// TIA Portal V17 program export: 1 tag tables, 0 data types, 2 data blocks, 7 code blocks (in call order from the OBs), 24 instance data blocks

VAR_GLOBAL   // PLC tag table "Default tag table"
   i_PB_RESET_BEZPIECZENSTWA AT %I0.0 : Bool;
   i_KURTYNA_ŚWIETLNA_OK AT %I0.1 : Bool;
   i_E_STOP_OK AT %I0.2 : Bool;
   i_PB_START AT %I0.3 : Bool;
   i_PB_STOP AT %I0.4 : Bool;
   i_SIŁOWNIK_ZACISKAJĄCY_UGÓRY AT %I0.5 : Bool;
   i_SIŁOWNIK_ZACISKAJĄCY_W_DOLE AT %I0.6 : Bool;
   "i_SIŁOWNIK NASTAWY_GŁĘBOKIE" AT %I0.7 : Bool;
   "i_SIŁOWNIK NASTAWY _PŁYTKIE" AT %I1.0 : Bool;
   i_SIŁOWNIK_ODBIORU_POZ_STÓŁ AT %I1.1 : Bool;
   i_SIŁOWNIK_ODBIORU_POZ_ZRZUT AT %I1.2 : Bool;
   i_CZUJNIK_POZYCJI_STOŁU AT %I1.3 : Bool;
   i_CZUJNIK_SZTUKI_OK AT %I1.4 : Bool;
   i_CZUJNIK_PŁYTKIE_PRZÓD AT %I1.5 : Bool;
   Axis_1_Drive_IN AT %I68.0 : "PD_TEL3_IN";
   q_GŁÓWNY_ZAWÓR_POWIETRZA_ON AT %Q0.0 : Bool;
   q_NIEBIESKA_LAMPKA_SAFETY AT %Q0.1 : Bool;
   q_SIŁOWNIK_ZACISKAJĄCY_DOL AT %Q0.2 : Bool;
   q_EJECTOR_VACUM AT %Q0.3 : Bool;
   q_SIŁOWNIK_ZMIANY_GŁĘBOKIE AT %Q0.4 : Bool;
   q_EJECTOR_BLOWOFF AT %Q0.5 : Bool;
   q_SIŁOWNIK_ODBIERAJĄCY_STÓŁ AT %Q0.6 : Bool;
   q_LED_LAMP AT %Q0.7 : Bool;
   q_REZERWA1 AT %Q1.0 : Bool;
   q_REZERWA2 AT %Q1.1 : Bool;
   q_CZERWONA_KOLUMNA_SYGNALIZACYJNA AT %Q8.0 : Bool;
   q_ZÓŁTA_KOLUMNA_SYGNALIZACYJNA AT %Q8.1 : Bool;
   q_ZIELONA_KOLUMNA_SYGNALIZACYJNA AT %Q8.2 : Bool;
   q_BUZZER_KOLUMNA_SYGNALIZACYJNA AT %Q8.3 : Bool;
   q_SAFETY_RELAY_RESET AT %Q8.4 : Bool;
   q_REZERWA4 AT %Q8.5 : Bool;
   q_REZERWA5 AT %Q8.6 : Bool;
   q_REZERWA6 AT %Q8.7 : Bool;
   Clock_Byte AT %MB0 : Byte;
   Clock_10Hz AT %M0.0 : Bool;
   Clock_5Hz AT %M0.1 : Bool;
   "Clock_2.5Hz" AT %M0.2 : Bool;
   Clock_2Hz AT %M0.3 : Bool;
   "Clock_1.25Hz" AT %M0.4 : Bool;
   Clock_1Hz AT %M0.5 : Bool;
   "Clock_0.625Hz" AT %M0.6 : Bool;
   "Clock_0.5Hz" AT %M0.7 : Bool;
   m_SAFETY_OK AT %M1.0 : Bool;
   m_AUTO_MODE AT %M1.1 : Bool;
   m_SERVO_READY AT %M1.2 : Bool;
   MAN_SIŁ_ZAG_GÓRA AT %M1.3 : Bool;
   MAN_SIŁ_ZAG_DÓŁ AT %M1.4 : Bool;
   MAN_SIŁ_NASTAWY_GŁĘBOKIE AT %M1.5 : Bool;
   MAN_SIŁ_NASTAWY_PŁYTKIE AT %M1.6 : Bool;
   MAN_SIŁ_ODBIOR_STÓŁ AT %M1.7 : Bool;
   MAN_SIŁ_ODBIOR_ZRZUT AT %M2.0 : Bool;
   MAN_JOG_STOL_FWD AT %M2.1 : Bool;
   MAN_JOG_STOL_BWD AT %M2.2 : Bool;
   MAN_POZYCJA_STÓŁ_FWD AT %M2.3 : Bool;
   MAN_POZYCJA_STÓŁ_BWD AT %M2.4 : Bool;
   MAN_EJECTOR_SSANIE AT %M2.5 : Bool;
   MAN_EJECTOR_PRZEDMUCH AT %M2.6 : Bool;
   TP_ZAPISZ_WARTOŚĆ_PRED AT %M2.7 : Bool;
   TP_ZAPISZ_WARTOŚĆ_CZASU_PRZEDMUCHU AT %M3.0 : Bool;
   TP_ZAPISZ_WARTOSC_CZASU_SSANIA AT %M3.1 : Bool;
   TP_AKT_PRED_STOŁU AT %MW4 : Int;
   TP_NOWA_PRED_STOŁU AT %MW6 : Int;
   TP_AKT_CZAS_PRZEDMUCHU AT %MD50 : DInt;
   TP_NOWY_CZAS_PRZEDMUCHU AT %MD54 : DInt;
   TP_AKT_CZAS_SSANIA AT %MD58 : DInt;
   TP_NOWY_CZAS_SSANIA AT %MD62 : DInt;
   TP_LICZNIK_CAŁKOWITY AT %MD16 : DInt;
   TP_LICZNIK_ZADANE AT %MD20 : DInt;
   TP_LICZNIK_WYKONANE AT %MD24 : DInt;
   TP_KASUJ_LICZNIK_ZADANE AT %M3.2 : Bool;
   TP_USTAW_LICZNIK_ZADANE AT %M3.3 : Bool;
   TP_KASUJ_LICZNIK_AKTUALNE AT %M3.4 : Bool;
   m_STOL_KAT_OBROTU AT %MW28 : Int;
   TP_LED_ZAŁĄCZ AT %M3.5 : Bool;
   m_SRV_STO_ON AT %M3.6 : Bool;
   TP_USTAW_CZAS_TAKTU AT %M3.7 : Bool;
   AUTO_NUMER_KROKU AT %MW30 : Int;
   AUTO_KROK_1_ZAŁADUNEK AT %M32.0 : Bool;
   AUTO_KROK_2_OBRÓT_USTAW_GŁĘBOKIE AT %M32.1 : Bool;
   AUTO_KROK_3_ROZŁADUNEK AT %M32.2 : Bool;
   AUTO_KROK_4_ZJAZD_GŁĘBOKIE AT %M32.3 : Bool;
   AUTO_KROK_5_OBRÓT_USTAW_PLYTKIE AT %M32.4 : Bool;
   "AUTO_KROK_6_ZJAZD GŁOWICY PŁYTKIE" AT %M32.5 : Bool;
   AUTO_SERVO_FWD AT %M34.0 : Bool;
   AUTO_SIŁOWNIK_ZACISKAJĄCY_DÓŁ AT %M34.1 : Bool;
   AUTO_SIŁOWNIK_ZACISKAJĄCY_GÓRA AT %M34.2 : Bool;
   AUTO_SIŁOWNIK_NASTAWY_GŁĘBOKIE AT %M34.3 : Bool;
   AUTO_SIŁOWNIK_NASTAWY_PŁYTKIE AT %M34.4 : Bool;
   AUTO_SIŁOWNIK_ODBIORU_STÓŁ AT %M34.5 : Bool;
   AUTO_SIŁOWNIK_ODBIORU_ZRZUT AT %M34.6 : Bool;
   AUTO_EJECTOR_SSANIE AT %M34.7 : Bool;
   AUTO_EJECTOR_PRZEDMUCH AT %M35.0 : Bool;
   AUTO_TAKT_OBRÓT AT %MW38 : Int;
   TP_TAKT_ZADANA AT %MW40 : Int;
   TEST_BIT AT %M100.2 : Bool;
   TP_LAMP_TEST AT %M43.1 : Bool;
   m_TRYB_RĘCZNY_MOŻLIWY AT %M42.0 : Bool;
   MAN_Q_SIŁ_ZAG_GÓRA AT %M42.1 : Bool;
   MAN_Q_SIŁ_ZAG_DÓŁ AT %M42.2 : Bool;
   MAN_Q_SIŁ_NAS_GŁĘBOKIE AT %M42.3 : Bool;
   MAN_Q_SIŁ_NAS_PLYTKIE AT %M42.4 : Bool;
   MAN_Q_SIŁ_ODB_ZRZUT AT %M42.6 : Bool;
   MAN_Q_EJECTOR_SSANIE AT %M42.7 : Bool;
   MAN_Q_SIŁ_ODB_STÓŁ AT %M42.5 : Bool;
   MAN_Q_EJECTOR_PRZEDMUCH AT %M43.0 : Bool;
   m_ALARM_ACTIVE AT %M43.2 : Bool;
   m_WARNING_ACTIVE AT %M43.3 : Bool;
   AUTO_KROK2_WARUNKI_OK AT %M43.4 : Bool;
   m_ZBOCZE_P_POZ_STOŁU AT %M43.5 : Bool;
   m_ZBOCZE_P_CZUJNIK_SZTUK AT %M43.6 : Bool;
   AUTO_KROK5_WARUNKI_OK AT %M43.7 : Bool;
   AUTO_KROK6_WARUNKI_OK AT %M44.0 : Bool;
   TP_SCREEN_NO AT %MW46 : Int;
   System_Byte AT %MB1000 : Byte;
   FirstScan AT %M1000.0 : Bool;
   DiagStatusUpdate AT %M1000.1 : Bool;
   AlwaysTRUE AT %M1000.2 : Bool;
   AlwaysFALSE AT %M1000.3 : Bool;
   AUTO_CZAS_PRZEDMUCHU_SEK AT %MD66 : DInt;
   AUTO_CZAS_SSANIA_SEK AT %MD68 : DInt;
   test_power_in_enbl AT %M200.0 : Bool;
   TP_BTN_SET_HOME_POS AT %M358.3 : Bool;
   "temp_to pos_fwd" AT %M358.4 : Bool;
   temp_czujnik_poz_stolu_puls AT %M358.5 : Bool;
   "temp_to pos_bwd" AT %M358.6 : Bool;
   m_table_is_home AT %M358.7 : Bool;
   test_1 AT %M359.0 : Bool;
   test_2 AT %M359.1 : Bool;
   test_3 AT %M359.2 : Bool;
   test_4 AT %M359.3 : Bool;
   test_5 AT %M359.4 : Bool;
   test_6 AT %M359.5 : Bool;
   test_7 AT %M359.6 : Bool;
   test_8 AT %M359.7 : Bool;
   test_9 AT %M360.0 : Bool;
   test_10 AT %M360.1 : Bool;
   test_11 AT %M360.2 : Bool;
   test_12 AT %M360.3 : Bool;
   test_13 AT %M360.4 : Bool;
   test_14 AT %M360.5 : Bool;
   test_15 AT %M360.6 : Bool;
   test_16 AT %M360.7 : Bool;
   Axis_1_Drive_OUT AT %Q68.0 : "PD_TEL3_OUT";
   m_no_collision_table AT %M361.0 : Bool;
   TP_USTAW_DELAY_SIŁ_ZAG AT %M361.1 : Bool;
   TP_USTAW_DELAY_SIŁ_ODB AT %M361.2 : Bool;
   m_auto_table_velocity AT %MD362 : Real;
   m_memo_cycle_start AT %M8.0 : Bool;
   m_cycle_auto_possible AT %M8.1 : Bool;
   m_zbocze_N_kurtyna AT %M8.2 : Bool;
   m_auto_table_start_pos AT %M8.3 : Bool;
   m_zbocze_P_pb_start AT %M8.4 : Bool;
   m_zbocze_P_licznik AT %M8.5 : Bool;
   m_zbocze_P_licznik2 AT %M8.6 : Bool;
   tp_table_home_ok AT %M8.7 : Bool;
   m_memo_czujnik_stol_takt AT %M9.0 : Bool;
   m_memo_turn_started AT %M9.1 : Bool;
   m_auto_tact_time_elapsed AT %M9.2 : Bool;
   m_zbocze_N_czuj_stoł AT %M9.3 : Bool;
   m_memo_time_tack_elapsed AT %M9.4 : Bool;
   "m_auto_to pos_fwd" AT %M9.5 : Bool;
   temp_calc_new_tact AT %MD10 : Real;
   tp_display_akt_tact_time AT %MD72 : Real;
   m_zbocze_N_ustaw_takt AT %M9.6 : Bool;
   m_ustaw_takt_puls AT %M9.7 : Bool;
   tp_display_akt_sucktion_time AT %MD76 : Real;
   m_zbocze_N_ustaw_czas_ssania AT %M14.0 : Bool;
   tp_display_akt_blow_time AT %MD80 : Real;
   tp_display_akt_delay_sił_zag AT %MD84 : Real;
   tp_display_akt_delay_sił_odb AT %MD88 : Real;
   "m_zbocze_N-_czas_przedmuchu" AT %M14.1 : Bool;
   m_zboczeN_ustaw_delay_zagn AT %M14.2 : Bool;
   m_zboczeN_ustaw_delay_odbioru AT %M14.3 : Bool;
   m_zbocze_P_ustaw_czas_przedm AT %M14.4 : Bool;
   m_zbocze_P_delay_sił_zagniatania AT %M14.5 : Bool;
   m_auto_siłownik_odb_stoł AT %M14.6 : Bool;
   m_delay_sił_odbioru_elapsed AT %M14.7 : Bool;
   m_auto_zezwolenie_ssanie AT %M15.0 : Bool;
   m_delay_ssanie_elapsed AT %M15.1 : Bool;
   m_auto_zezwolenie_przedmuch AT %M15.2 : Bool;
   m_delay_przedmuch_elapsed AT %M15.3 : Bool;
   m_manual_mode AT %M15.4 : Bool;
   m_zbocze_czujnik_stołP2 AT %M15.5 : Bool;
   Flaga_nr_gniazda AT %M15.6 : Bool;
   m_zboczeN_zakon_przedmuch AT %M15.7 : Bool;
   m_potw_zakonczenia_rozł AT %M32.6 : Bool;
   m_zboczP_nowy_cykl_siłownika AT %M32.7 : Bool;
   m_memo_zboczeP_poz_odb AT %M33.0 : Bool;
   m_zbocze1 AT %M33.1 : Bool;
   m_zbocze2 AT %M33.2 : Bool;
   m_zbocze3 AT %M33.3 : Bool;
   m_auto_cycle_glebokie_gniazdo AT %M33.4 : Bool;
   m_auto_zmien_na_glebokie AT %M33.5 : Bool;
   m_zbocze4 AT %M33.6 : Bool;
   m_cycle5 AT %M33.7 : Bool;
   m_auto_sił_zagniatania_dol AT %M35.1 : Bool;
   m_auto_delay_zag_elapsed AT %M35.2 : Bool;
   m_stol_memo AT %M35.3 : Bool;
   m_zbocze5 AT %M35.4 : Bool;
   m_memo_kurtynaP AT %M35.5 : Bool;
   m_kurtyna_podczas_obrotu AT %M35.6 : Bool;
   m_sztuka_OK AT %M35.7 : Bool;
   m_obrót_krok AT %M36.0 : Bool;
   m_czujnik_ok AT %M36.1 : Bool;
   m_wykonano_zadana_ilosc AT %M36.2 : Bool;
   "m_powiadomienie_o zakonczeniu" AT %M36.3 : Bool;
   m_add_qty_cmpl AT %M36.4 : Bool;
   m_zboczeN_sztuki_OK AT %M36.5 : Bool;
   m_dodano AT %M36.6 : Bool;
   test1 AT %M36.7 : Bool;
END_VAR

DATA_BLOCK "proces_value"   // DB12
{ S7_Optimized_Access := 'TRUE' }
VERSION : 0.1
// stored: AutoNumber true, DBAccessibleFromOPCUA true, IsOnlyStoredInLoadMemory false, IsRetainMemResEnabled false, IsWriteProtectedInAS false, MemoryReserve 100
   VAR RETAIN
      db_tp_akt_pred_stołu : Real := 50.0;
   END_VAR
   VAR
      db_tp_nowa_pred_stołu : Real;
   END_VAR
   VAR RETAIN
      db_tp_akt_takt_stołu : Time := T#7S;
   END_VAR
   VAR
      db_tp_nowy_takt_stołu : Real;
   END_VAR
   VAR RETAIN
      db_tp_akt_czas_ssania : Time := T#1S;
   END_VAR
   VAR
      db_tp_nowy_czas_ssania : Real;
   END_VAR
   VAR RETAIN
      "db_tp_akt_czas przedmuchu" : Time := T#1S;
   END_VAR
   VAR
      db_tp_nowy_czas_przedmuchu : Real;
   END_VAR
   VAR RETAIN
      db_tp_akt_delay_sił_zag : Time := T#100MS;
   END_VAR
   VAR
      db_tp_nowy_delay_sił_zag : Real;
   END_VAR
   VAR RETAIN
      db_tp_akt_delay_sił_odbioru_stoł : Time := T#1S;
   END_VAR
   VAR
      db_tp_nowy_delay_sił_odbioru_stoł : Real;
   END_VAR
   VAR RETAIN
      db_licznik_calkowity : DInt;
      db_licznik_zadane : DInt;
      db_licznik_wykonane : DInt;
      db_aktualne_gniazdo : Int;
      db_auto_table_velocity : Real := 0.5;
   END_VAR
BEGIN
END_DATA_BLOCK

DATA_BLOCK "reference_values"   // DB26
{ S7_Optimized_Access := 'TRUE' }
VERSION : 0.1
// stored: AutoNumber true, DBAccessibleFromOPCUA true, IsOnlyStoredInLoadMemory false, IsRetainMemResEnabled false, IsWriteProtectedInAS false, MemoryReserve 100
   VAR RETAIN
      ref1_takt_stołu : Time := T#7S;
      ref1_pred_stolu : Real := 50.0;
      ref1_czas_ssania : Time := T#1S;
      ref1_czas_przedmuchu : Time := T#1S;
      ref1_delay_sił_zag_dół : Time := T#100MS;
   END_VAR
   VAR
      ref1_delay_sił_odb_stol : Time := T#1S;
   END_VAR
BEGIN
END_DATA_BLOCK

ORGANIZATION_BLOCK "Main"   // OB1, LAD, ProgramCycle
TITLE = "Main Program Sweep (Cycle)"
{ S7_Optimized_Access := 'TRUE' }
VERSION : 0.1
// stored: AutoNumber true, IsIECCheckEnabled false, SetENOAutomatically false
   VAR_INPUT
      Initial_Call : Bool;   // Initial call of this OB
      Remanence : Bool;   // =True, if remanent data are available
   END_VAR
BEGIN

REGION Network 1: AUTO MODE SET FROM HMI
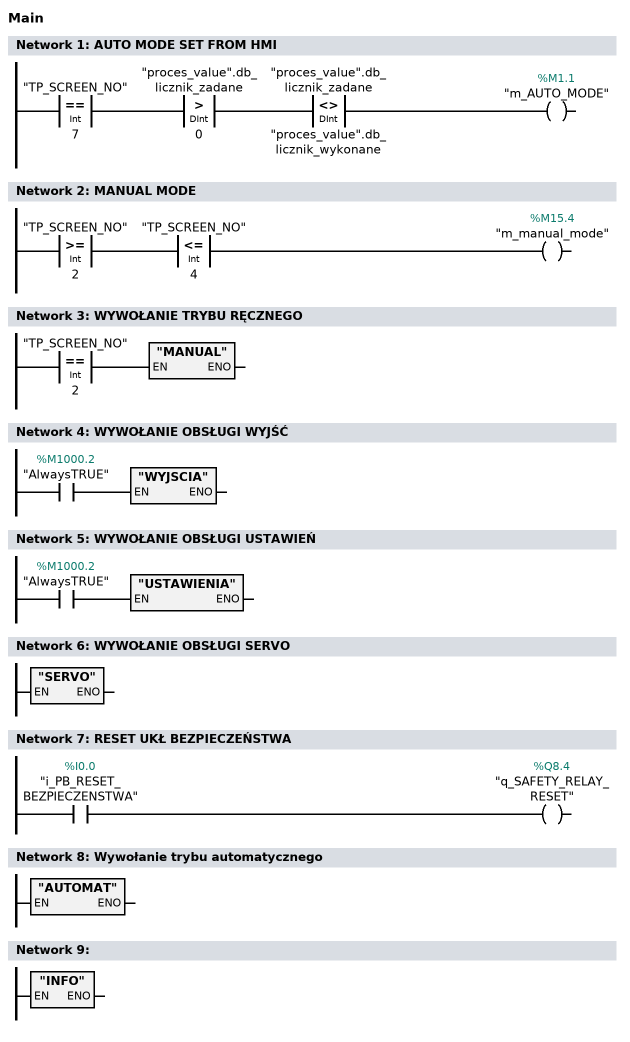
   RUNG wire#powerrail
      { S7_Templates := "SrcType := Int" } EQ_Contact(in1 := "TP_SCREEN_NO", in2 := 7)
      { S7_Templates := "SrcType := DInt" } GT_Contact(in1 := "proces_value".db_licznik_zadane, in2 := 0)
      { S7_Templates := "SrcType := DInt" } NE_Contact(in1 := "proces_value".db_licznik_zadane, in2 := "proces_value".db_licznik_wykonane)
      Coil( "m_AUTO_MODE" )
   END_RUNG
   // the same network as SCL:
   "m_AUTO_MODE" := ("TP_SCREEN_NO" = 7) AND ("proces_value".db_licznik_zadane > 0) AND ("proces_value".db_licznik_zadane <> "proces_value".db_licznik_wykonane);
END_REGION

REGION Network 2: MANUAL MODE
   RUNG wire#powerrail
      { S7_Templates := "SrcType := Int" } GE_Contact(in1 := "TP_SCREEN_NO", in2 := 2)
      { S7_Templates := "SrcType := Int" } LE_Contact(in1 := "TP_SCREEN_NO", in2 := 4)
      Coil( "m_manual_mode" )
   END_RUNG
   // the same network as SCL:
   "m_manual_mode" := ("TP_SCREEN_NO" >= 2) AND ("TP_SCREEN_NO" <= 4);
END_REGION

REGION Network 3: WYWOŁANIE TRYBU RĘCZNEGO
   RUNG wire#powerrail
      { S7_Templates := "SrcType := Int" } EQ_Contact(in1 := "TP_SCREEN_NO", in2 := 2)
      "MANUAL"()
   END_RUNG
   // the same network as SCL:
   IF "TP_SCREEN_NO" = 2 THEN "MANUAL"(); END_IF;
END_REGION

REGION Network 4: WYWOŁANIE OBSŁUGI WYJŚĆ
   RUNG wire#powerrail
      Contact( "AlwaysTRUE" )
      "WYJSCIA"()
   END_RUNG
   // the same network as SCL:
   IF "AlwaysTRUE" THEN "WYJSCIA"(); END_IF;
END_REGION

REGION Network 5: WYWOŁANIE OBSŁUGI USTAWIEŃ
   RUNG wire#powerrail
      Contact( "AlwaysTRUE" )
      "USTAWIENIA"()
   END_RUNG
   // the same network as SCL:
   IF "AlwaysTRUE" THEN "USTAWIENIA"(); END_IF;
END_REGION

REGION Network 6: WYWOŁANIE OBSŁUGI SERVO
   RUNG wire#powerrail
      "SERVO"()
   END_RUNG
   // the same network as SCL:
   "SERVO"();
END_REGION

REGION Network 7: RESET UKŁ BEZPIECZEŃSTWA
   RUNG wire#powerrail
      Contact( "i_PB_RESET_BEZPIECZENSTWA" )
      Coil( "q_SAFETY_RELAY_RESET" )
   END_RUNG
   // the same network as SCL:
   "q_SAFETY_RELAY_RESET" := "i_PB_RESET_BEZPIECZENSTWA";
END_REGION

REGION Network 8: Wywołanie trybu automatycznego
   RUNG wire#powerrail
      "AUTOMAT"()
   END_RUNG
   // the same network as SCL:
   "AUTOMAT"();
END_REGION

REGION Network 9
   RUNG wire#powerrail
      "INFO"()
   END_RUNG
   // the same network as SCL:
   "INFO"();
END_REGION
END_ORGANIZATION_BLOCK

FUNCTION "MANUAL" : Void   // FC1, LAD
{ S7_Optimized_Access := 'TRUE' }
VERSION : 0.1
// stored: AutoNumber true, IsIECCheckEnabled false, SetENOAutomatically false, UDAEnableTagReadback false
   VAR_TEMP   // added for the SCL form of the ladder/FBD networks
      _w1 : Bool;
   END_VAR
BEGIN

REGION Network 1: WARUNKI DLA TRYBU RĘCZNEGO
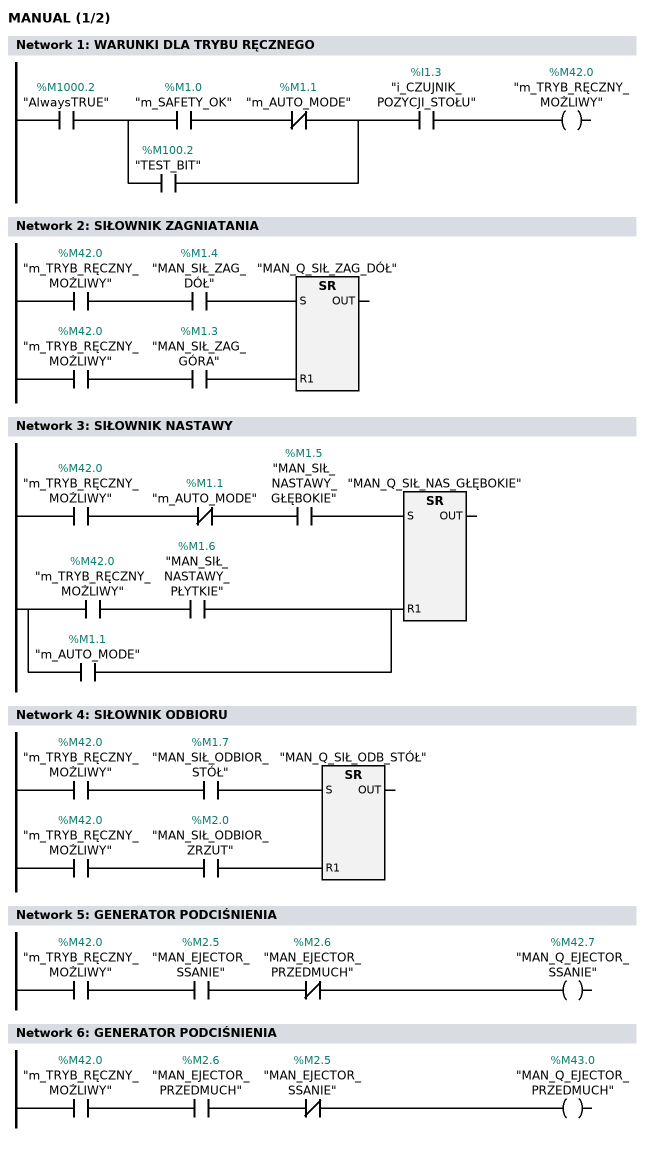
   RUNG wire#powerrail
      Contact( "AlwaysTRUE" )
      wire#w1
      Contact( "m_SAFETY_OK" )
      I_Contact( "m_AUTO_MODE" )
      wire#w2
      Contact( "i_CZUJNIK_POZYCJI_STOŁU" )
      Coil( "m_TRYB_RĘCZNY_MOŻLIWY" )
   END_RUNG
   RUNG wire#w1
      Contact( "TEST_BIT" )
   END_RUNG wire#w2
   // the same network as SCL:
   "m_TRYB_RĘCZNY_MOŻLIWY" := "AlwaysTRUE" AND (("m_SAFETY_OK" AND NOT "m_AUTO_MODE") OR "TEST_BIT") AND "i_CZUJNIK_POZYCJI_STOŁU";
END_REGION

REGION Network 2: SIŁOWNIK ZAGNIATANIA
   RUNG wire#powerrail
      Contact( "m_TRYB_RĘCZNY_MOŻLIWY" )
      Contact( "MAN_SIŁ_ZAG_DÓŁ" )
      S_SR(operand := "MAN_Q_SIŁ_ZAG_DÓŁ", r1 := wire#w1)
   END_RUNG
   RUNG wire#powerrail
      Contact( "m_TRYB_RĘCZNY_MOŻLIWY" )
      Contact( "MAN_SIŁ_ZAG_GÓRA" )
   END_RUNG wire#w1
   // the same network as SCL:
   IF "m_TRYB_RĘCZNY_MOŻLIWY" AND "MAN_SIŁ_ZAG_DÓŁ" THEN
       "MAN_Q_SIŁ_ZAG_DÓŁ" := TRUE;   // SR flip-flop
   END_IF;
   IF "m_TRYB_RĘCZNY_MOŻLIWY" AND "MAN_SIŁ_ZAG_GÓRA" THEN "MAN_Q_SIŁ_ZAG_DÓŁ" := FALSE; END_IF;
END_REGION

REGION Network 3: SIŁOWNIK NASTAWY
   RUNG wire#powerrail
      Contact( "m_TRYB_RĘCZNY_MOŻLIWY" )
      I_Contact( "m_AUTO_MODE" )
      Contact( "MAN_SIŁ_NASTAWY_GŁĘBOKIE" )
      S_SR(operand := "MAN_Q_SIŁ_NAS_GŁĘBOKIE", r1 := wire#w1)
   END_RUNG
   RUNG wire#powerrail
      Contact( "m_TRYB_RĘCZNY_MOŻLIWY" )
      Contact( "MAN_SIŁ_NASTAWY_PŁYTKIE" )
   END_RUNG wire#w1
   RUNG wire#powerrail
      Contact( "m_AUTO_MODE" )
   END_RUNG wire#w1
   // the same network as SCL:
   IF "m_TRYB_RĘCZNY_MOŻLIWY" AND NOT "m_AUTO_MODE" AND "MAN_SIŁ_NASTAWY_GŁĘBOKIE" THEN
       "MAN_Q_SIŁ_NAS_GŁĘBOKIE" := TRUE;   // SR flip-flop
   END_IF;
   IF ("m_TRYB_RĘCZNY_MOŻLIWY" AND "MAN_SIŁ_NASTAWY_PŁYTKIE") OR "m_AUTO_MODE" THEN
       "MAN_Q_SIŁ_NAS_GŁĘBOKIE" := FALSE;
   END_IF;
END_REGION

REGION Network 4: SIŁOWNIK ODBIORU
   RUNG wire#powerrail
      Contact( "m_TRYB_RĘCZNY_MOŻLIWY" )
      Contact( "MAN_SIŁ_ODBIOR_STÓŁ" )
      S_SR(operand := "MAN_Q_SIŁ_ODB_STÓŁ", r1 := wire#w1)
   END_RUNG
   RUNG wire#powerrail
      Contact( "m_TRYB_RĘCZNY_MOŻLIWY" )
      Contact( "MAN_SIŁ_ODBIOR_ZRZUT" )
   END_RUNG wire#w1
   // the same network as SCL:
   IF "m_TRYB_RĘCZNY_MOŻLIWY" AND "MAN_SIŁ_ODBIOR_STÓŁ" THEN
       "MAN_Q_SIŁ_ODB_STÓŁ" := TRUE;   // SR flip-flop
   END_IF;
   IF "m_TRYB_RĘCZNY_MOŻLIWY" AND "MAN_SIŁ_ODBIOR_ZRZUT" THEN "MAN_Q_SIŁ_ODB_STÓŁ" := FALSE; END_IF;
END_REGION

REGION Network 5: GENERATOR PODCIŚNIENIA
   RUNG wire#powerrail
      Contact( "m_TRYB_RĘCZNY_MOŻLIWY" )
      Contact( "MAN_EJECTOR_SSANIE" )
      I_Contact( "MAN_EJECTOR_PRZEDMUCH" )
      Coil( "MAN_Q_EJECTOR_SSANIE" )
   END_RUNG
   // the same network as SCL:
   "MAN_Q_EJECTOR_SSANIE" := "m_TRYB_RĘCZNY_MOŻLIWY" AND "MAN_EJECTOR_SSANIE" AND NOT "MAN_EJECTOR_PRZEDMUCH";
END_REGION

REGION Network 6: GENERATOR PODCIŚNIENIA
   RUNG wire#powerrail
      Contact( "m_TRYB_RĘCZNY_MOŻLIWY" )
      Contact( "MAN_EJECTOR_PRZEDMUCH" )
      I_Contact( "MAN_EJECTOR_SSANIE" )
      Coil( "MAN_Q_EJECTOR_PRZEDMUCH" )
   END_RUNG
   // the same network as SCL:
   "MAN_Q_EJECTOR_PRZEDMUCH" := "m_TRYB_RĘCZNY_MOŻLIWY" AND "MAN_EJECTOR_PRZEDMUCH" AND NOT "MAN_EJECTOR_SSANIE";
END_REGION

REGION Network 7: RUCHY RECZNE STOŁU DO POZYCJI FWD
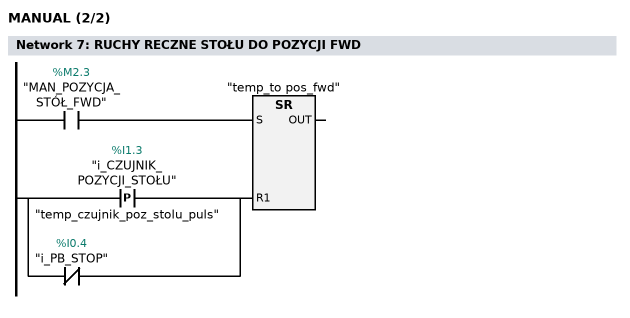
   RUNG wire#powerrail
      Contact( "MAN_POZYCJA_STÓŁ_FWD" )
      S_SR(operand := "temp_to pos_fwd", r1 := wire#w1)
   END_RUNG
   RUNG wire#powerrail
      P_Contact(operand := "i_CZUJNIK_POZYCJI_STOŁU", bit := "temp_czujnik_poz_stolu_puls")
   END_RUNG wire#w1
   RUNG wire#powerrail
      I_Contact( "i_PB_STOP" )
   END_RUNG wire#w1
   // the same network as SCL:
   #_w1 := "i_CZUJNIK_POZYCJI_STOŁU" AND NOT "temp_czujnik_poz_stolu_puls";   // rising edge of "i_CZUJNIK_POZYCJI_STOŁU"
   "temp_czujnik_poz_stolu_puls" := "i_CZUJNIK_POZYCJI_STOŁU";
   IF "MAN_POZYCJA_STÓŁ_FWD" THEN
       "temp_to pos_fwd" := TRUE;   // SR flip-flop
   END_IF;
   IF #_w1 OR NOT "i_PB_STOP" THEN "temp_to pos_fwd" := FALSE; END_IF;
END_REGION
END_FUNCTION

FUNCTION "WYJSCIA" : Void   // FC2, LAD
{ S7_Optimized_Access := 'TRUE' }
VERSION : 0.1
// stored: AutoNumber true, IsIECCheckEnabled false, SetENOAutomatically false, UDAEnableTagReadback false
BEGIN

REGION Network 1: SAFETY OK
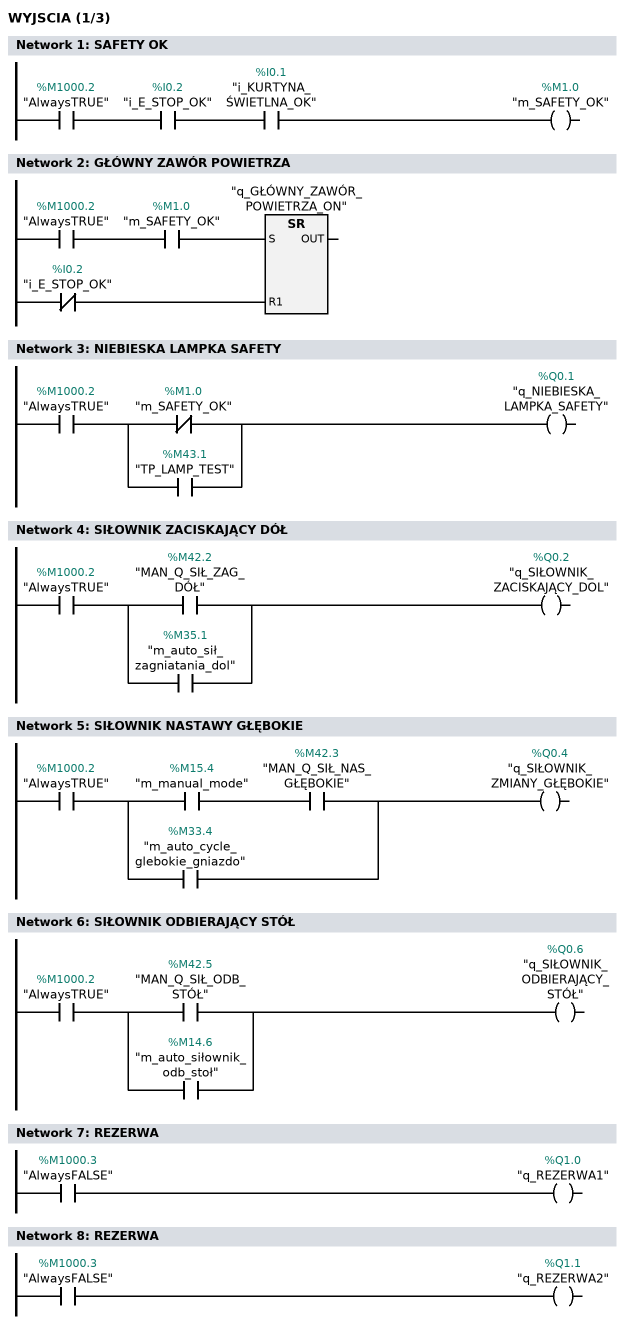
   RUNG wire#powerrail
      Contact( "AlwaysTRUE" )
      Contact( "i_E_STOP_OK" )
      Contact( "i_KURTYNA_ŚWIETLNA_OK" )
      Coil( "m_SAFETY_OK" )
   END_RUNG
   // the same network as SCL:
   "m_SAFETY_OK" := "AlwaysTRUE" AND "i_E_STOP_OK" AND "i_KURTYNA_ŚWIETLNA_OK";
END_REGION

REGION Network 2: GŁÓWNY ZAWÓR POWIETRZA
   RUNG wire#powerrail
      Contact( "AlwaysTRUE" )
      Contact( "m_SAFETY_OK" )
      S_SR(operand := "q_GŁÓWNY_ZAWÓR_POWIETRZA_ON", r1 := wire#w1)
   END_RUNG
   RUNG wire#powerrail
      I_Contact( "i_E_STOP_OK" )
   END_RUNG wire#w1
   // the same network as SCL:
   IF "AlwaysTRUE" AND "m_SAFETY_OK" THEN
       "q_GŁÓWNY_ZAWÓR_POWIETRZA_ON" := TRUE;   // SR flip-flop
   END_IF;
   IF NOT "i_E_STOP_OK" THEN "q_GŁÓWNY_ZAWÓR_POWIETRZA_ON" := FALSE; END_IF;
END_REGION

REGION Network 3: NIEBIESKA LAMPKA SAFETY
   RUNG wire#powerrail
      Contact( "AlwaysTRUE" )
      wire#w1
      I_Contact( "m_SAFETY_OK" )
      wire#w2
      Coil( "q_NIEBIESKA_LAMPKA_SAFETY" )
   END_RUNG
   RUNG wire#w1
      Contact( "TP_LAMP_TEST" )
   END_RUNG wire#w2
   // the same network as SCL:
   "q_NIEBIESKA_LAMPKA_SAFETY" := "AlwaysTRUE" AND (NOT "m_SAFETY_OK" OR "TP_LAMP_TEST");
END_REGION

REGION Network 4: SIŁOWNIK ZACISKAJĄCY DÓŁ
   RUNG wire#powerrail
      Contact( "AlwaysTRUE" )
      wire#w1
      Contact( "MAN_Q_SIŁ_ZAG_DÓŁ" )
      wire#w2
      Coil( "q_SIŁOWNIK_ZACISKAJĄCY_DOL" )
   END_RUNG
   RUNG wire#w1
      Contact( "m_auto_sił_zagniatania_dol" )
   END_RUNG wire#w2
   // the same network as SCL:
   "q_SIŁOWNIK_ZACISKAJĄCY_DOL" := "AlwaysTRUE" AND ("MAN_Q_SIŁ_ZAG_DÓŁ" OR "m_auto_sił_zagniatania_dol");
END_REGION

REGION Network 5: SIŁOWNIK NASTAWY GŁĘBOKIE
   RUNG wire#powerrail
      Contact( "AlwaysTRUE" )
      wire#w1
      Contact( "m_manual_mode" )
      Contact( "MAN_Q_SIŁ_NAS_GŁĘBOKIE" )
      wire#w2
      Coil( "q_SIŁOWNIK_ZMIANY_GŁĘBOKIE" )
   END_RUNG
   RUNG wire#w1
      Contact( "m_auto_cycle_glebokie_gniazdo" )
   END_RUNG wire#w2
   // the same network as SCL:
   "q_SIŁOWNIK_ZMIANY_GŁĘBOKIE" := "AlwaysTRUE" AND (("m_manual_mode" AND "MAN_Q_SIŁ_NAS_GŁĘBOKIE") OR "m_auto_cycle_glebokie_gniazdo");
END_REGION

REGION Network 6: SIŁOWNIK ODBIERAJĄCY STÓŁ
   RUNG wire#powerrail
      Contact( "AlwaysTRUE" )
      wire#w1
      Contact( "MAN_Q_SIŁ_ODB_STÓŁ" )
      wire#w2
      Coil( "q_SIŁOWNIK_ODBIERAJĄCY_STÓŁ" )
   END_RUNG
   RUNG wire#w1
      Contact( "m_auto_siłownik_odb_stoł" )
   END_RUNG wire#w2
   // the same network as SCL:
   "q_SIŁOWNIK_ODBIERAJĄCY_STÓŁ" := "AlwaysTRUE" AND ("MAN_Q_SIŁ_ODB_STÓŁ" OR "m_auto_siłownik_odb_stoł");
END_REGION

REGION Network 7: REZERWA
   RUNG wire#powerrail
      Contact( "AlwaysFALSE" )
      Coil( "q_REZERWA1" )
   END_RUNG
   // the same network as SCL:
   "q_REZERWA1" := "AlwaysFALSE";
END_REGION

REGION Network 8: REZERWA
   RUNG wire#powerrail
      Contact( "AlwaysFALSE" )
      Coil( "q_REZERWA2" )
   END_RUNG
   // the same network as SCL:
   "q_REZERWA2" := "AlwaysFALSE";
END_REGION

REGION Network 9: EJECTOR SSANIE
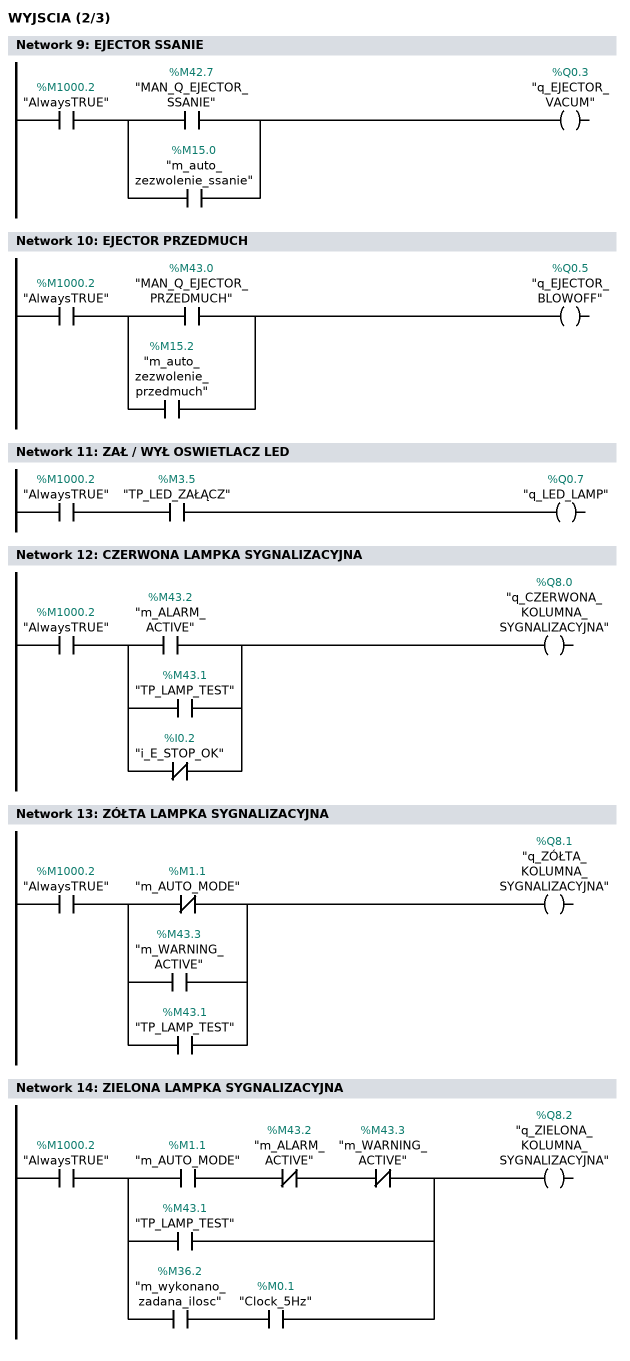
   RUNG wire#powerrail
      Contact( "AlwaysTRUE" )
      wire#w1
      Contact( "MAN_Q_EJECTOR_SSANIE" )
      wire#w2
      Coil( "q_EJECTOR_VACUM" )
   END_RUNG
   RUNG wire#w1
      Contact( "m_auto_zezwolenie_ssanie" )
   END_RUNG wire#w2
   // the same network as SCL:
   "q_EJECTOR_VACUM" := "AlwaysTRUE" AND ("MAN_Q_EJECTOR_SSANIE" OR "m_auto_zezwolenie_ssanie");
END_REGION

REGION Network 10: EJECTOR PRZEDMUCH
   RUNG wire#powerrail
      Contact( "AlwaysTRUE" )
      wire#w1
      Contact( "MAN_Q_EJECTOR_PRZEDMUCH" )
      wire#w2
      Coil( "q_EJECTOR_BLOWOFF" )
   END_RUNG
   RUNG wire#w1
      Contact( "m_auto_zezwolenie_przedmuch" )
   END_RUNG wire#w2
   // the same network as SCL:
   "q_EJECTOR_BLOWOFF" := "AlwaysTRUE" AND ("MAN_Q_EJECTOR_PRZEDMUCH" OR "m_auto_zezwolenie_przedmuch");
END_REGION

REGION Network 11: ZAŁ / WYŁ OSWIETLACZ LED
   RUNG wire#powerrail
      Contact( "AlwaysTRUE" )
      Contact( "TP_LED_ZAŁĄCZ" )
      Coil( "q_LED_LAMP" )
   END_RUNG
   // the same network as SCL:
   "q_LED_LAMP" := "AlwaysTRUE" AND "TP_LED_ZAŁĄCZ";
END_REGION

REGION Network 12: CZERWONA LAMPKA SYGNALIZACYJNA
   RUNG wire#powerrail
      Contact( "AlwaysTRUE" )
      wire#w1
      Contact( "m_ALARM_ACTIVE" )
      wire#w2
      Coil( "q_CZERWONA_KOLUMNA_SYGNALIZACYJNA" )
   END_RUNG
   RUNG wire#w1
      Contact( "TP_LAMP_TEST" )
   END_RUNG wire#w2
   RUNG wire#w1
      I_Contact( "i_E_STOP_OK" )
   END_RUNG wire#w2
   // the same network as SCL:
   "q_CZERWONA_KOLUMNA_SYGNALIZACYJNA" := "AlwaysTRUE" AND ("m_ALARM_ACTIVE" OR "TP_LAMP_TEST" OR NOT "i_E_STOP_OK");
END_REGION

REGION Network 13: ZÓŁTA LAMPKA SYGNALIZACYJNA
   RUNG wire#powerrail
      Contact( "AlwaysTRUE" )
      wire#w1
      I_Contact( "m_AUTO_MODE" )
      wire#w2
      Coil( "q_ZÓŁTA_KOLUMNA_SYGNALIZACYJNA" )
   END_RUNG
   RUNG wire#w1
      Contact( "m_WARNING_ACTIVE" )
   END_RUNG wire#w2
   RUNG wire#w1
      Contact( "TP_LAMP_TEST" )
   END_RUNG wire#w2
   // the same network as SCL:
   "q_ZÓŁTA_KOLUMNA_SYGNALIZACYJNA" := "AlwaysTRUE" AND (NOT "m_AUTO_MODE" OR "m_WARNING_ACTIVE" OR "TP_LAMP_TEST");
END_REGION

REGION Network 14: ZIELONA LAMPKA SYGNALIZACYJNA
   RUNG wire#powerrail
      Contact( "AlwaysTRUE" )
      wire#w1
      Contact( "m_AUTO_MODE" )
      I_Contact( "m_ALARM_ACTIVE" )
      I_Contact( "m_WARNING_ACTIVE" )
      wire#w2
      Coil( "q_ZIELONA_KOLUMNA_SYGNALIZACYJNA" )
   END_RUNG
   RUNG wire#w1
      Contact( "TP_LAMP_TEST" )
   END_RUNG wire#w2
   RUNG wire#w1
      Contact( "m_wykonano_zadana_ilosc" )
      Contact( "Clock_5Hz" )
   END_RUNG wire#w2
   // the same network as SCL:
   "q_ZIELONA_KOLUMNA_SYGNALIZACYJNA" := "AlwaysTRUE" AND (("m_AUTO_MODE" AND NOT "m_ALARM_ACTIVE" AND NOT "m_WARNING_ACTIVE") OR "TP_LAMP_TEST" OR ("m_wykonano_zadana_ilosc" AND "Clock_5Hz"));
END_REGION

REGION Network 15: BUZZER KOLUMNA SYGNALIZACYJNA
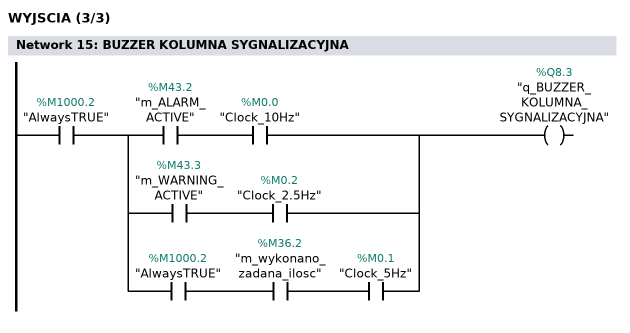
   RUNG wire#powerrail
      Contact( "AlwaysTRUE" )
      wire#w1
      Contact( "m_ALARM_ACTIVE" )
      Contact( "Clock_10Hz" )
      wire#w2
      Coil( "q_BUZZER_KOLUMNA_SYGNALIZACYJNA" )
   END_RUNG
   RUNG wire#w1
      Contact( "m_WARNING_ACTIVE" )
      Contact( "Clock_2.5Hz" )
   END_RUNG wire#w2
   RUNG wire#w1
      Contact( "AlwaysTRUE" )
      Contact( "m_wykonano_zadana_ilosc" )
      Contact( "Clock_5Hz" )
   END_RUNG wire#w2
   // the same network as SCL:
   "q_BUZZER_KOLUMNA_SYGNALIZACYJNA" := "AlwaysTRUE" AND (("m_ALARM_ACTIVE" AND "Clock_10Hz") OR ("m_WARNING_ACTIVE" AND "Clock_2.5Hz") OR ("AlwaysTRUE" AND "m_wykonano_zadana_ilosc" AND "Clock_5Hz"));
END_REGION
END_FUNCTION

FUNCTION "USTAWIENIA" : Void   // FC3, LAD
{ S7_Optimized_Access := 'TRUE' }
VERSION : 0.1
// stored: AutoNumber true, IsIECCheckEnabled false, SetENOAutomatically false, UDAEnableTagReadback false
   VAR_TEMP
      temp_calc_new_tact2 : DInt;
      temp_calc_3 : DInt;
      temp_calc4 : Real;
      temp_calc5 : DInt;
      temp_calc6 : DInt;
      m_zboczeP_ustaw_czas_ssania : Bool;
      temp_calc7 : Real;
      temp_calc8 : Real;
      temp_calc9 : Real;
      temp_calc10 : DInt;
      temp_calc11 : DInt;
      temp_calc12 : Real;
      temp_calc13 : Real;
      temp_calc14 : DInt;
      temp_calc15 : DInt;
      temp_calc16 : Real;
      temp_calc17 : Real;
      temp_calc18 : DInt;
      temp_calc19 : DInt;
      temp_calc20 : Real;
      m_zboczeN_ustaw_delay_zag : Bool;
      m_zboczeN_ustaw_delay_odb : Bool;
      m_zbocze_P_ustaw_delay_odbior : Bool;
   END_VAR
   VAR_TEMP   // added for the SCL form of the ladder/FBD networks
      _w1 : Bool;
      _w2 : Bool;
      _w3 : Bool;
      _w4 : Bool;
      _w5 : Bool;
      _w6 : Bool;
   END_VAR
BEGIN

REGION Network 1: KASOWANIE LICZNIKÓW ZADANYCH SZTUK I WYKONANYCH
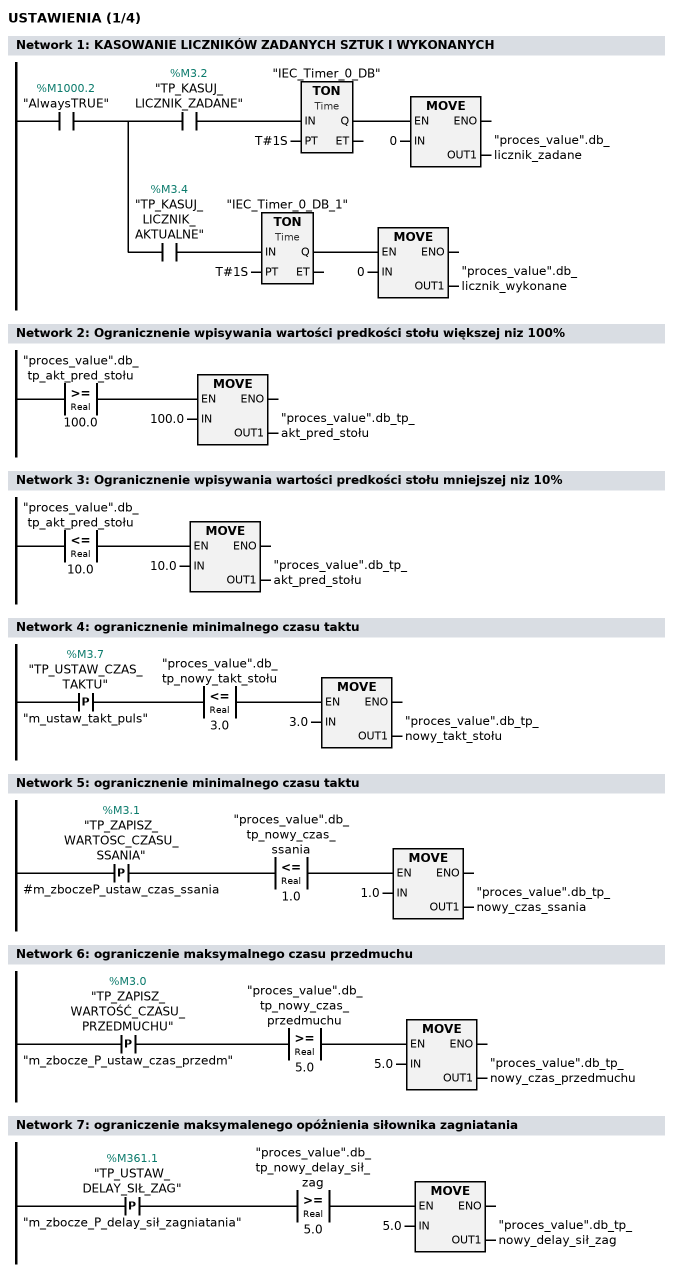
   RUNG wire#powerrail
      Contact( "AlwaysTRUE" )
      wire#w1
      Contact( "TP_KASUJ_LICZNIK_ZADANE" )
      { S7_Templates := "time_type := Time" } "IEC_Timer_0_DB".TON(pt := T#1S, et =>)
      Move(in := 0, out1 => "proces_value".db_licznik_zadane)
   END_RUNG
   RUNG wire#w1
      Contact( "TP_KASUJ_LICZNIK_AKTUALNE" )
      { S7_Templates := "time_type := Time" } "IEC_Timer_0_DB_1".TON(pt := T#1S, et =>)
      Move(in := 0, out1 => "proces_value".db_licznik_wykonane)
   END_RUNG
   // the same network as SCL:
   "IEC_Timer_0_DB".TON(IN := "AlwaysTRUE" AND "TP_KASUJ_LICZNIK_ZADANE", PT := T#1S);
   IF "IEC_Timer_0_DB".Q THEN "proces_value".db_licznik_zadane := 0; END_IF;
   "IEC_Timer_0_DB_1".TON(IN := "AlwaysTRUE" AND "TP_KASUJ_LICZNIK_AKTUALNE", PT := T#1S);
   IF "IEC_Timer_0_DB_1".Q THEN "proces_value".db_licznik_wykonane := 0; END_IF;
END_REGION

REGION Network 2: Ogranicznenie wpisywania wartości predkości stołu większej niz 100%
   RUNG wire#powerrail
      { S7_Templates := "SrcType := Real" } GE_Contact(in1 := "proces_value".db_tp_akt_pred_stołu, in2 := 100.0)
      Move(in := 100.0, out1 => "proces_value".db_tp_akt_pred_stołu)
   END_RUNG
   // the same network as SCL:
   IF "proces_value".db_tp_akt_pred_stołu >= 100.0 THEN "proces_value".db_tp_akt_pred_stołu := 100.0; END_IF;
END_REGION

REGION Network 3: Ogranicznenie wpisywania wartości predkości stołu mniejszej niz 10%
   RUNG wire#powerrail
      { S7_Templates := "SrcType := Real" } LE_Contact(in1 := "proces_value".db_tp_akt_pred_stołu, in2 := 10.0)
      Move(in := 10.0, out1 => "proces_value".db_tp_akt_pred_stołu)
   END_RUNG
   // the same network as SCL:
   IF "proces_value".db_tp_akt_pred_stołu <= 10.0 THEN "proces_value".db_tp_akt_pred_stołu := 10.0; END_IF;
END_REGION

REGION Network 4: ogranicznenie minimalnego czasu taktu
   RUNG wire#powerrail
      P_Contact(operand := "TP_USTAW_CZAS_TAKTU", bit := "m_ustaw_takt_puls")
      { S7_Templates := "SrcType := Real" } LE_Contact(in1 := "proces_value".db_tp_nowy_takt_stołu, in2 := 3.0)
      Move(in := 3.0, out1 => "proces_value".db_tp_nowy_takt_stołu)
   END_RUNG
   // the same network as SCL:
   #_w1 := "TP_USTAW_CZAS_TAKTU" AND NOT "m_ustaw_takt_puls";   // rising edge of "TP_USTAW_CZAS_TAKTU"
   "m_ustaw_takt_puls" := "TP_USTAW_CZAS_TAKTU";
   IF #_w1 AND ("proces_value".db_tp_nowy_takt_stołu <= 3.0) THEN
       "proces_value".db_tp_nowy_takt_stołu := 3.0;
   END_IF;
END_REGION

REGION Network 5: ogranicznenie minimalnego czasu taktu
   RUNG wire#powerrail
      P_Contact(operand := "TP_ZAPISZ_WARTOSC_CZASU_SSANIA", bit := #m_zboczeP_ustaw_czas_ssania)
      { S7_Templates := "SrcType := Real" } LE_Contact(in1 := "proces_value".db_tp_nowy_czas_ssania, in2 := 1.0)
      Move(in := 1.0, out1 => "proces_value".db_tp_nowy_czas_ssania)
   END_RUNG
   // the same network as SCL:
   #_w1 := "TP_ZAPISZ_WARTOSC_CZASU_SSANIA" AND NOT #m_zboczeP_ustaw_czas_ssania;   // rising edge of "TP_ZAPISZ_WARTOSC_CZASU_SSANIA"
   #m_zboczeP_ustaw_czas_ssania := "TP_ZAPISZ_WARTOSC_CZASU_SSANIA";
   IF #_w1 AND ("proces_value".db_tp_nowy_czas_ssania <= 1.0) THEN
       "proces_value".db_tp_nowy_czas_ssania := 1.0;
   END_IF;
END_REGION

REGION Network 6: ograniczenie maksymalnego czasu przedmuchu
   RUNG wire#powerrail
      P_Contact(operand := "TP_ZAPISZ_WARTOŚĆ_CZASU_PRZEDMUCHU", bit := "m_zbocze_P_ustaw_czas_przedm")
      { S7_Templates := "SrcType := Real" } GE_Contact(in1 := "proces_value".db_tp_nowy_czas_przedmuchu, in2 := 5.0)
      Move(in := 5.0, out1 => "proces_value".db_tp_nowy_czas_przedmuchu)
   END_RUNG
   // the same network as SCL:
   #_w1 := "TP_ZAPISZ_WARTOŚĆ_CZASU_PRZEDMUCHU" AND NOT "m_zbocze_P_ustaw_czas_przedm";   // rising edge of "TP_ZAPISZ_WARTOŚĆ_CZASU_PRZEDMUCHU"
   "m_zbocze_P_ustaw_czas_przedm" := "TP_ZAPISZ_WARTOŚĆ_CZASU_PRZEDMUCHU";
   IF #_w1 AND ("proces_value".db_tp_nowy_czas_przedmuchu >= 5.0) THEN
       "proces_value".db_tp_nowy_czas_przedmuchu := 5.0;
   END_IF;
END_REGION

REGION Network 7: ograniczenie maksymalenego opóżnienia siłownika zagniatania
   RUNG wire#powerrail
      P_Contact(operand := "TP_USTAW_DELAY_SIŁ_ZAG", bit := "m_zbocze_P_delay_sił_zagniatania")
      { S7_Templates := "SrcType := Real" } GE_Contact(in1 := "proces_value".db_tp_nowy_delay_sił_zag, in2 := 5.0)
      Move(in := 5.0, out1 => "proces_value".db_tp_nowy_delay_sił_zag)
   END_RUNG
   // the same network as SCL:
   #_w1 := "TP_USTAW_DELAY_SIŁ_ZAG" AND NOT "m_zbocze_P_delay_sił_zagniatania";   // rising edge of "TP_USTAW_DELAY_SIŁ_ZAG"
   "m_zbocze_P_delay_sił_zagniatania" := "TP_USTAW_DELAY_SIŁ_ZAG";
   IF #_w1 AND ("proces_value".db_tp_nowy_delay_sił_zag >= 5.0) THEN
       "proces_value".db_tp_nowy_delay_sił_zag := 5.0;
   END_IF;
END_REGION

REGION Network 8: ograniczenie maksymalenego opóżnienia siłownika odbioru
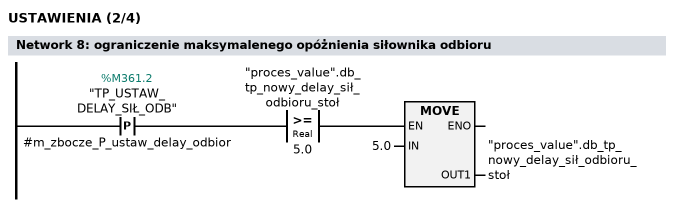
   RUNG wire#powerrail
      P_Contact(operand := "TP_USTAW_DELAY_SIŁ_ODB", bit := #m_zbocze_P_ustaw_delay_odbior)
      { S7_Templates := "SrcType := Real" } GE_Contact(in1 := "proces_value".db_tp_nowy_delay_sił_odbioru_stoł, in2 := 5.0)
      Move(in := 5.0, out1 => "proces_value".db_tp_nowy_delay_sił_odbioru_stoł)
   END_RUNG
   // the same network as SCL:
   #_w1 := "TP_USTAW_DELAY_SIŁ_ODB" AND NOT #m_zbocze_P_ustaw_delay_odbior;   // rising edge of "TP_USTAW_DELAY_SIŁ_ODB"
   #m_zbocze_P_ustaw_delay_odbior := "TP_USTAW_DELAY_SIŁ_ODB";
   IF #_w1 AND ("proces_value".db_tp_nowy_delay_sił_odbioru_stoł >= 5.0) THEN
       "proces_value".db_tp_nowy_delay_sił_odbioru_stoł := 5.0;
   END_IF;
END_REGION

REGION Network 9: OBSŁUGA LICZNIKÓW I TIMERÓW
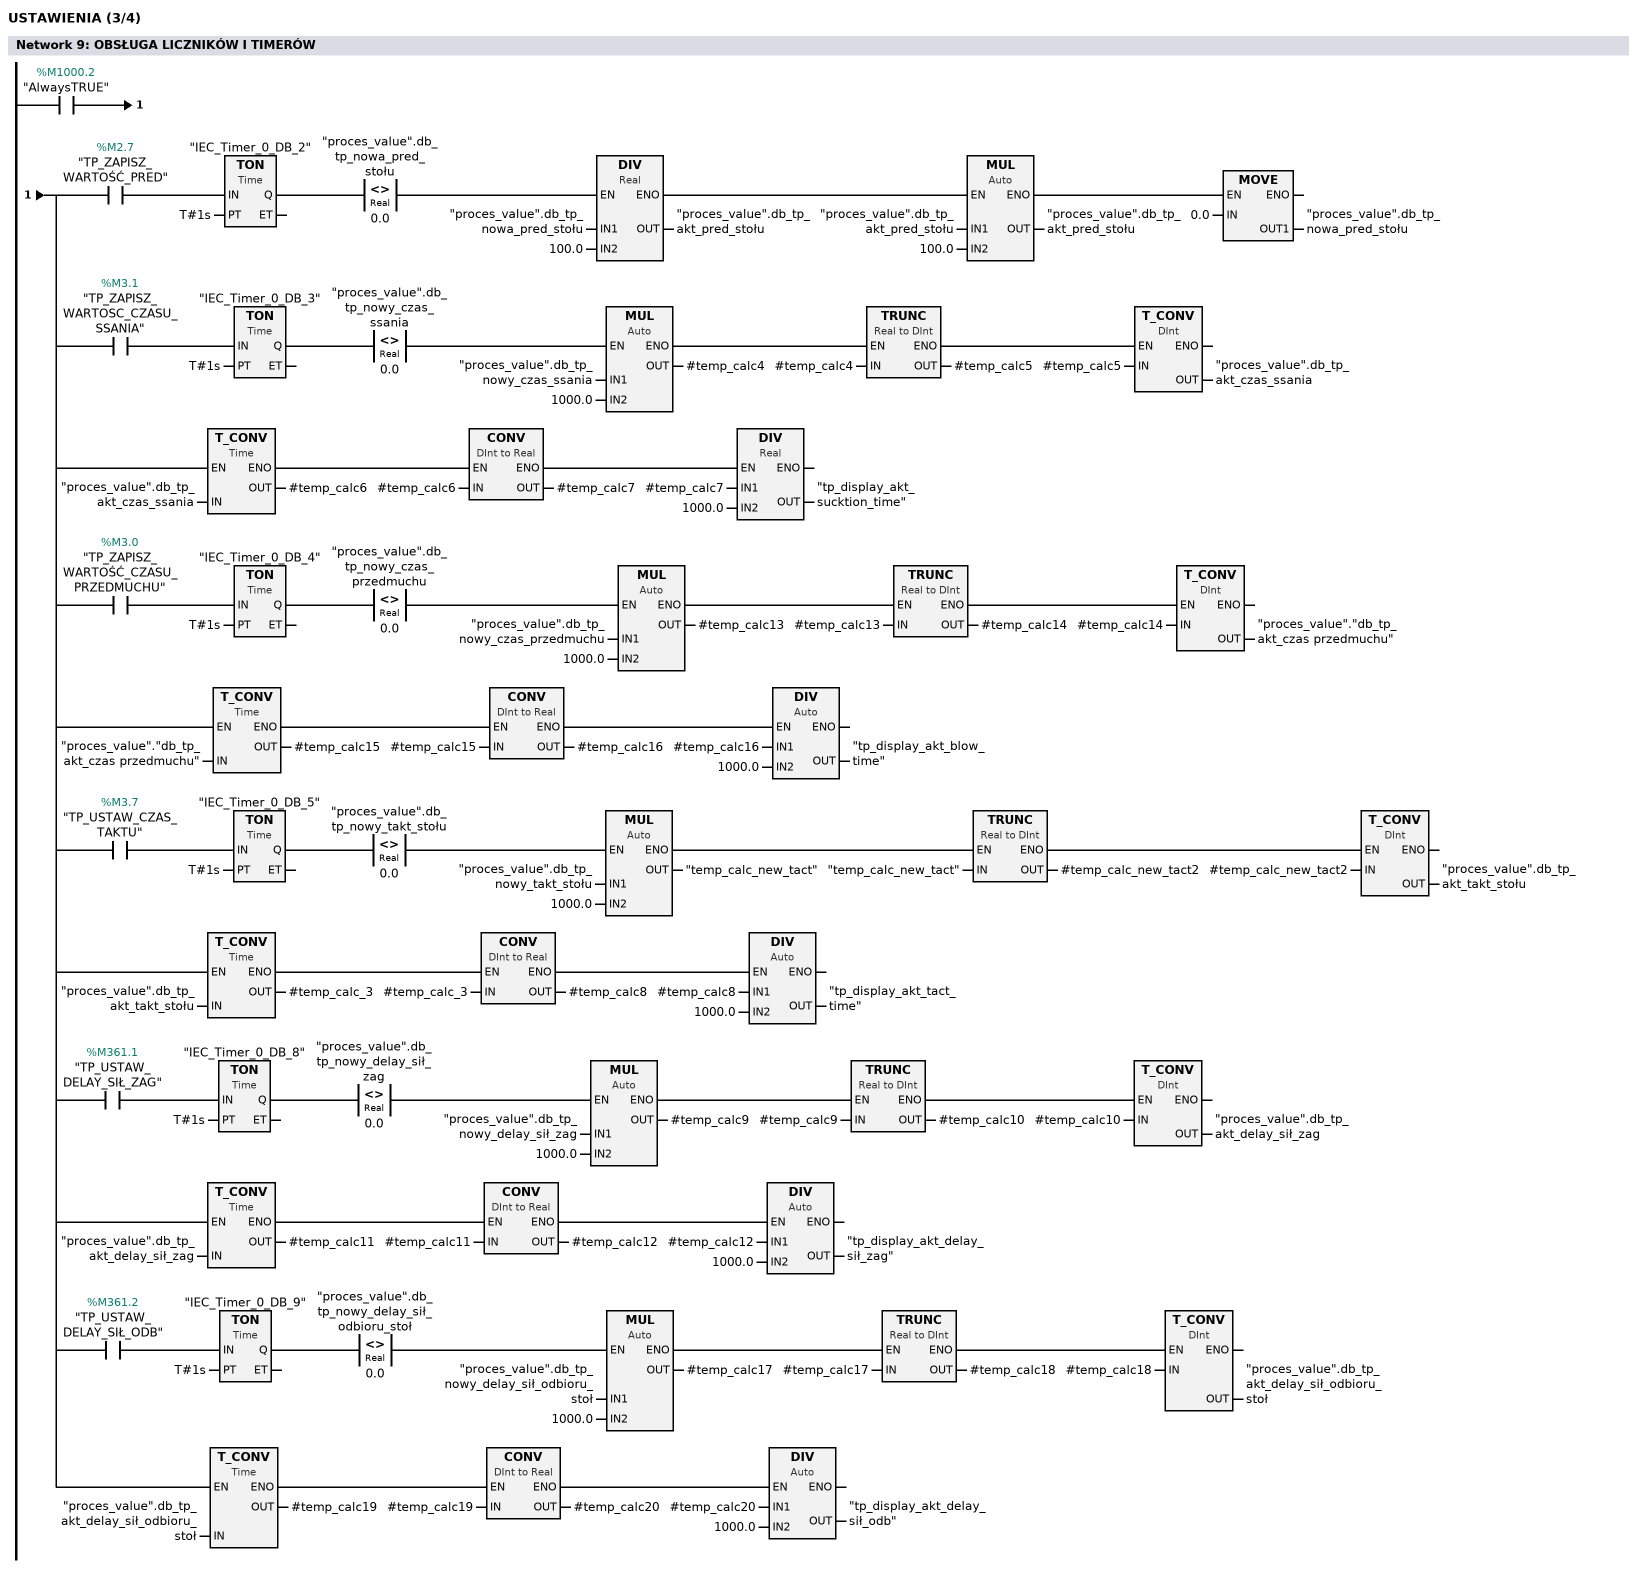
   RUNG wire#powerrail
      Contact( "AlwaysTRUE" )
      wire#w1
      Contact( "TP_ZAPISZ_WARTOŚĆ_PRED" )
      { S7_Templates := "time_type := Time" } "IEC_Timer_0_DB_2".TON(pt := T#1s, et =>)
      { S7_Templates := "SrcType := Real" } NE_Contact(in1 := "proces_value".db_tp_nowa_pred_stołu, in2 := 0.0)
      { S7_Templates := "SrcType := Real" } Div(in1 := "proces_value".db_tp_nowa_pred_stołu, in2 := 100.0, out => "proces_value".db_tp_akt_pred_stołu)
      Mul(in1 := "proces_value".db_tp_akt_pred_stołu, in2 := 100.0, out => "proces_value".db_tp_akt_pred_stołu)
      Move(in := 0.0, out1 => "proces_value".db_tp_nowa_pred_stołu)
   END_RUNG
   RUNG wire#w1
      Contact( "TP_ZAPISZ_WARTOSC_CZASU_SSANIA" )
      { S7_Templates := "time_type := Time" } "IEC_Timer_0_DB_3".TON(pt := T#1s, et =>)
      { S7_Templates := "SrcType := Real" } NE_Contact(in1 := "proces_value".db_tp_nowy_czas_ssania, in2 := 0.0)
      Mul(in1 := "proces_value".db_tp_nowy_czas_ssania, in2 := 1000.0, out => #temp_calc4)
      { S7_Templates := "[SrcType := Real, DestType := DInt]" } Trunc(in := #temp_calc4, out => #temp_calc5)
      { S7_Templates := "[src_type := DInt, dest_type := Time]" } T_CONV(IN := #temp_calc5, OUT => "proces_value".db_tp_akt_czas_ssania)
   END_RUNG
   RUNG wire#w1
      { S7_Templates := "[src_type := Time, dest_type := DInt]" } T_CONV(IN := "proces_value".db_tp_akt_czas_ssania, OUT => #temp_calc6)
      { S7_Templates := "[SrcType := DInt, DestType := Real]" } Convert(in := #temp_calc6, out => #temp_calc7)
      { S7_Templates := "SrcType := Real" } Div(in1 := #temp_calc7, in2 := 1000.0, out => "tp_display_akt_sucktion_time")
   END_RUNG
   RUNG wire#w1
      Contact( "TP_ZAPISZ_WARTOŚĆ_CZASU_PRZEDMUCHU" )
      { S7_Templates := "time_type := Time" } "IEC_Timer_0_DB_4".TON(pt := T#1s, et =>)
      { S7_Templates := "SrcType := Real" } NE_Contact(in1 := "proces_value".db_tp_nowy_czas_przedmuchu, in2 := 0.0)
      Mul(in1 := "proces_value".db_tp_nowy_czas_przedmuchu, in2 := 1000.0, out => #temp_calc13)
      { S7_Templates := "[SrcType := Real, DestType := DInt]" } Trunc(in := #temp_calc13, out => #temp_calc14)
      { S7_Templates := "[src_type := DInt, dest_type := Time]" } T_CONV(IN := #temp_calc14, OUT => "proces_value"."db_tp_akt_czas przedmuchu")
   END_RUNG
   RUNG wire#w1
      { S7_Templates := "[src_type := Time, dest_type := DInt]" } T_CONV(IN := "proces_value"."db_tp_akt_czas przedmuchu", OUT => #temp_calc15)
      { S7_Templates := "[SrcType := DInt, DestType := Real]" } Convert(in := #temp_calc15, out => #temp_calc16)
      Div(in1 := #temp_calc16, in2 := 1000.0, out => "tp_display_akt_blow_time")
   END_RUNG
   RUNG wire#w1
      Contact( "TP_USTAW_CZAS_TAKTU" )
      { S7_Templates := "time_type := Time" } "IEC_Timer_0_DB_5".TON(pt := T#1s, et =>)
      { S7_Templates := "SrcType := Real" } NE_Contact(in1 := "proces_value".db_tp_nowy_takt_stołu, in2 := 0.0)
      Mul(in1 := "proces_value".db_tp_nowy_takt_stołu, in2 := 1000.0, out => "temp_calc_new_tact")
      { S7_Templates := "[SrcType := Real, DestType := DInt]" } Trunc(in := "temp_calc_new_tact", out => #temp_calc_new_tact2)
      { S7_Templates := "[src_type := DInt, dest_type := Time]" } T_CONV(IN := #temp_calc_new_tact2, OUT => "proces_value".db_tp_akt_takt_stołu)
   END_RUNG
   RUNG wire#w1
      { S7_Templates := "[src_type := Time, dest_type := DInt]" } T_CONV(IN := "proces_value".db_tp_akt_takt_stołu, OUT => #temp_calc_3)
      { S7_Templates := "[SrcType := DInt, DestType := Real]" } Convert(in := #temp_calc_3, out => #temp_calc8)
      Div(in1 := #temp_calc8, in2 := 1000.0, out => "tp_display_akt_tact_time")
   END_RUNG
   RUNG wire#w1
      Contact( "TP_USTAW_DELAY_SIŁ_ZAG" )
      { S7_Templates := "time_type := Time" } "IEC_Timer_0_DB_8".TON(pt := T#1s, et =>)
      { S7_Templates := "SrcType := Real" } NE_Contact(in1 := "proces_value".db_tp_nowy_delay_sił_zag, in2 := 0.0)
      Mul(in1 := "proces_value".db_tp_nowy_delay_sił_zag, in2 := 1000.0, out => #temp_calc9)
      { S7_Templates := "[SrcType := Real, DestType := DInt]" } Trunc(in := #temp_calc9, out => #temp_calc10)
      { S7_Templates := "[src_type := DInt, dest_type := Time]" } T_CONV(IN := #temp_calc10, OUT => "proces_value".db_tp_akt_delay_sił_zag)
   END_RUNG
   RUNG wire#w1
      { S7_Templates := "[src_type := Time, dest_type := DInt]" } T_CONV(IN := "proces_value".db_tp_akt_delay_sił_zag, OUT => #temp_calc11)
      { S7_Templates := "[SrcType := DInt, DestType := Real]" } Convert(in := #temp_calc11, out => #temp_calc12)
      Div(in1 := #temp_calc12, in2 := 1000.0, out => "tp_display_akt_delay_sił_zag")
   END_RUNG
   RUNG wire#w1
      Contact( "TP_USTAW_DELAY_SIŁ_ODB" )
      { S7_Templates := "time_type := Time" } "IEC_Timer_0_DB_9".TON(pt := T#1s, et =>)
      { S7_Templates := "SrcType := Real" } NE_Contact(in1 := "proces_value".db_tp_nowy_delay_sił_odbioru_stoł, in2 := 0.0)
      Mul(in1 := "proces_value".db_tp_nowy_delay_sił_odbioru_stoł, in2 := 1000.0, out => #temp_calc17)
      { S7_Templates := "[SrcType := Real, DestType := DInt]" } Trunc(in := #temp_calc17, out => #temp_calc18)
      { S7_Templates := "[src_type := DInt, dest_type := Time]" } T_CONV(IN := #temp_calc18, OUT => "proces_value".db_tp_akt_delay_sił_odbioru_stoł)
   END_RUNG
   RUNG wire#w1
      { S7_Templates := "[src_type := Time, dest_type := DInt]" } T_CONV(IN := "proces_value".db_tp_akt_delay_sił_odbioru_stoł, OUT => #temp_calc19)
      { S7_Templates := "[SrcType := DInt, DestType := Real]" } Convert(in := #temp_calc19, out => #temp_calc20)
      Div(in1 := #temp_calc20, in2 := 1000.0, out => "tp_display_akt_delay_sił_odb")
   END_RUNG
   // the same network as SCL:
   "IEC_Timer_0_DB_2".TON(IN := "AlwaysTRUE" AND "TP_ZAPISZ_WARTOŚĆ_PRED", PT := T#1s);
   IF "IEC_Timer_0_DB_2".Q AND ("proces_value".db_tp_nowa_pred_stołu <> 0.0) THEN
       "proces_value".db_tp_akt_pred_stołu := "proces_value".db_tp_nowa_pred_stołu / 100.0;
       "proces_value".db_tp_akt_pred_stołu := "proces_value".db_tp_akt_pred_stołu * 100.0;
       "proces_value".db_tp_nowa_pred_stołu := 0.0;
   END_IF;
   "IEC_Timer_0_DB_3".TON(IN := "AlwaysTRUE" AND "TP_ZAPISZ_WARTOSC_CZASU_SSANIA", PT := T#1s);
   IF "IEC_Timer_0_DB_3".Q AND ("proces_value".db_tp_nowy_czas_ssania <> 0.0) THEN
       #temp_calc4 := "proces_value".db_tp_nowy_czas_ssania * 1000.0;
       #temp_calc5 := TRUNC(#temp_calc4);
   END_IF;
   #_w1 := "AlwaysTRUE";
   IF "IEC_Timer_0_DB_3".Q AND ("proces_value".db_tp_nowy_czas_ssania <> 0.0) THEN
       T_CONV(IN := #temp_calc5, OUT => "proces_value".db_tp_akt_czas_ssania);
   END_IF;
   T_CONV(EN := #_w1, IN := "proces_value".db_tp_akt_czas_ssania, OUT => #temp_calc6, ENO => #_w2);
   IF #_w2 THEN
       #temp_calc7 := DINT_TO_REAL(#temp_calc6);
       "tp_display_akt_sucktion_time" := #temp_calc7 / 1000.0;
   END_IF;
   "IEC_Timer_0_DB_4".TON(IN := #_w1 AND "TP_ZAPISZ_WARTOŚĆ_CZASU_PRZEDMUCHU", PT := T#1s);
   IF "IEC_Timer_0_DB_4".Q AND ("proces_value".db_tp_nowy_czas_przedmuchu <> 0.0) THEN
       #temp_calc13 := "proces_value".db_tp_nowy_czas_przedmuchu * 1000.0;
       #temp_calc14 := TRUNC(#temp_calc13);
       T_CONV(IN := #temp_calc14, OUT => "proces_value"."db_tp_akt_czas przedmuchu");
   END_IF;
   T_CONV(EN := #_w1, IN := "proces_value"."db_tp_akt_czas przedmuchu", OUT => #temp_calc15, ENO => #_w3);
   IF #_w3 THEN
       #temp_calc16 := DINT_TO_REAL(#temp_calc15);
       "tp_display_akt_blow_time" := #temp_calc16 / 1000.0;
   END_IF;
   "IEC_Timer_0_DB_5".TON(IN := #_w1 AND "TP_USTAW_CZAS_TAKTU", PT := T#1s);
   IF "IEC_Timer_0_DB_5".Q AND ("proces_value".db_tp_nowy_takt_stołu <> 0.0) THEN
       "temp_calc_new_tact" := "proces_value".db_tp_nowy_takt_stołu * 1000.0;
       #temp_calc_new_tact2 := TRUNC("temp_calc_new_tact");
       T_CONV(IN := #temp_calc_new_tact2, OUT => "proces_value".db_tp_akt_takt_stołu);
   END_IF;
   T_CONV(EN := #_w1, IN := "proces_value".db_tp_akt_takt_stołu, OUT => #temp_calc_3, ENO => #_w4);
   IF #_w4 THEN
       #temp_calc8 := DINT_TO_REAL(#temp_calc_3);
       "tp_display_akt_tact_time" := #temp_calc8 / 1000.0;
   END_IF;
   "IEC_Timer_0_DB_8".TON(IN := #_w1 AND "TP_USTAW_DELAY_SIŁ_ZAG", PT := T#1s);
   IF "IEC_Timer_0_DB_8".Q AND ("proces_value".db_tp_nowy_delay_sił_zag <> 0.0) THEN
       #temp_calc9 := "proces_value".db_tp_nowy_delay_sił_zag * 1000.0;
       #temp_calc10 := TRUNC(#temp_calc9);
       T_CONV(IN := #temp_calc10, OUT => "proces_value".db_tp_akt_delay_sił_zag);
   END_IF;
   T_CONV(EN := #_w1, IN := "proces_value".db_tp_akt_delay_sił_zag, OUT => #temp_calc11, ENO => #_w5);
   IF #_w5 THEN
       #temp_calc12 := DINT_TO_REAL(#temp_calc11);
       "tp_display_akt_delay_sił_zag" := #temp_calc12 / 1000.0;
   END_IF;
   "IEC_Timer_0_DB_9".TON(IN := #_w1 AND "TP_USTAW_DELAY_SIŁ_ODB", PT := T#1s);
   IF "IEC_Timer_0_DB_9".Q AND ("proces_value".db_tp_nowy_delay_sił_odbioru_stoł <> 0.0) THEN
       #temp_calc17 := "proces_value".db_tp_nowy_delay_sił_odbioru_stoł * 1000.0;
       #temp_calc18 := TRUNC(#temp_calc17);
       T_CONV(IN := #temp_calc18, OUT => "proces_value".db_tp_akt_delay_sił_odbioru_stoł);
   END_IF;
   T_CONV(EN := #_w1, IN := "proces_value".db_tp_akt_delay_sił_odbioru_stoł, OUT => #temp_calc19, ENO => #_w6);
   IF #_w6 THEN
       #temp_calc20 := DINT_TO_REAL(#temp_calc19);
       "tp_display_akt_delay_sił_odb" := #temp_calc20 / 1000.0;
   END_IF;
END_REGION

REGION Network 10: podswietlenie przycisku po ustawieniu gniazda płytkiego jako 1
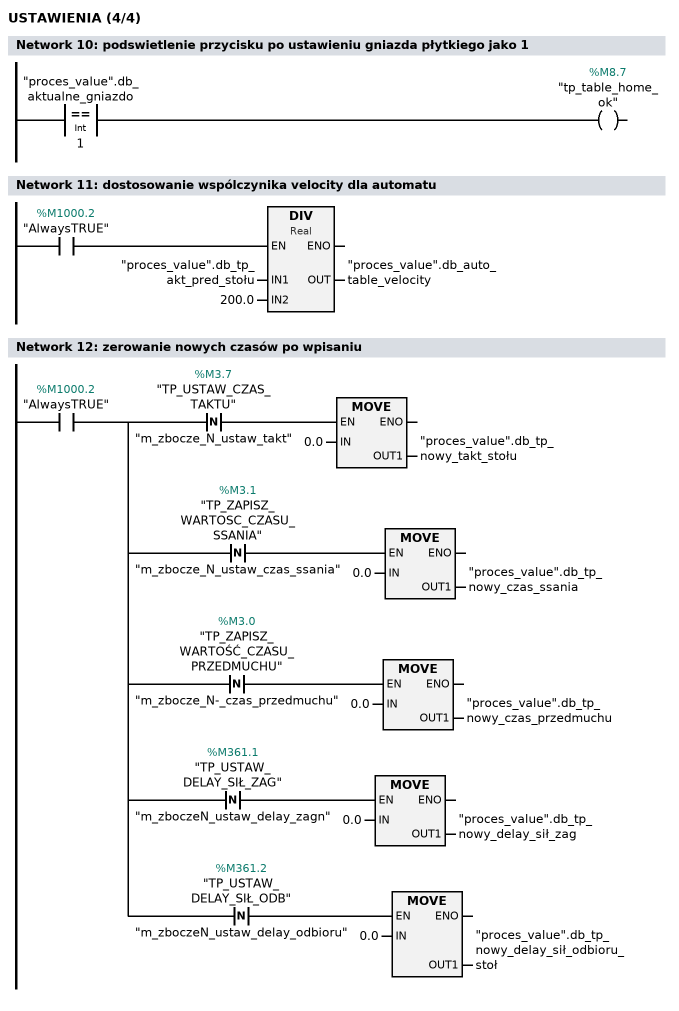
   RUNG wire#powerrail
      { S7_Templates := "SrcType := Int" } EQ_Contact(in1 := "proces_value".db_aktualne_gniazdo, in2 := 1)
      Coil( "tp_table_home_ok" )
   END_RUNG
   // the same network as SCL:
   "tp_table_home_ok" := "proces_value".db_aktualne_gniazdo = 1;
END_REGION

REGION Network 11: dostosowanie wspólczynika velocity dla automatu
   RUNG wire#powerrail
      Contact( "AlwaysTRUE" )
      { S7_Templates := "SrcType := Real" } Div(in1 := "proces_value".db_tp_akt_pred_stołu, in2 := 200.0, out => "proces_value".db_auto_table_velocity)
   END_RUNG
   // the same network as SCL:
   IF "AlwaysTRUE" THEN
       "proces_value".db_auto_table_velocity := "proces_value".db_tp_akt_pred_stołu / 200.0;
   END_IF;
END_REGION

REGION Network 12: zerowanie nowych czasów po wpisaniu
   RUNG wire#powerrail
      Contact( "AlwaysTRUE" )
      wire#w1
      N_Contact(operand := "TP_USTAW_CZAS_TAKTU", bit := "m_zbocze_N_ustaw_takt")
      Move(in := 0.0, out1 => "proces_value".db_tp_nowy_takt_stołu)
   END_RUNG
   RUNG wire#w1
      N_Contact(operand := "TP_ZAPISZ_WARTOSC_CZASU_SSANIA", bit := "m_zbocze_N_ustaw_czas_ssania")
      Move(in := 0.0, out1 => "proces_value".db_tp_nowy_czas_ssania)
   END_RUNG
   RUNG wire#w1
      N_Contact(operand := "TP_ZAPISZ_WARTOŚĆ_CZASU_PRZEDMUCHU", bit := "m_zbocze_N-_czas_przedmuchu")
      Move(in := 0.0, out1 => "proces_value".db_tp_nowy_czas_przedmuchu)
   END_RUNG
   RUNG wire#w1
      N_Contact(operand := "TP_USTAW_DELAY_SIŁ_ZAG", bit := "m_zboczeN_ustaw_delay_zagn")
      Move(in := 0.0, out1 => "proces_value".db_tp_nowy_delay_sił_zag)
   END_RUNG
   RUNG wire#w1
      N_Contact(operand := "TP_USTAW_DELAY_SIŁ_ODB", bit := "m_zboczeN_ustaw_delay_odbioru")
      Move(in := 0.0, out1 => "proces_value".db_tp_nowy_delay_sił_odbioru_stoł)
   END_RUNG
   // the same network as SCL:
   #_w1 := "AlwaysTRUE" AND NOT "TP_USTAW_CZAS_TAKTU" AND "m_zbocze_N_ustaw_takt";   // falling edge of "TP_USTAW_CZAS_TAKTU"
   "m_zbocze_N_ustaw_takt" := "TP_USTAW_CZAS_TAKTU";
   IF #_w1 THEN "proces_value".db_tp_nowy_takt_stołu := 0.0; END_IF;
   #_w2 := "AlwaysTRUE" AND NOT "TP_ZAPISZ_WARTOSC_CZASU_SSANIA" AND "m_zbocze_N_ustaw_czas_ssania";   // falling edge of "TP_ZAPISZ_WARTOSC_CZASU_SSANIA"
   "m_zbocze_N_ustaw_czas_ssania" := "TP_ZAPISZ_WARTOSC_CZASU_SSANIA";
   IF #_w2 THEN "proces_value".db_tp_nowy_czas_ssania := 0.0; END_IF;
   #_w3 := "AlwaysTRUE" AND NOT "TP_ZAPISZ_WARTOŚĆ_CZASU_PRZEDMUCHU" AND "m_zbocze_N-_czas_przedmuchu";   // falling edge of "TP_ZAPISZ_WARTOŚĆ_CZASU_PRZEDMUCHU"
   "m_zbocze_N-_czas_przedmuchu" := "TP_ZAPISZ_WARTOŚĆ_CZASU_PRZEDMUCHU";
   IF #_w3 THEN "proces_value".db_tp_nowy_czas_przedmuchu := 0.0; END_IF;
   #_w4 := "AlwaysTRUE" AND NOT "TP_USTAW_DELAY_SIŁ_ZAG" AND "m_zboczeN_ustaw_delay_zagn";   // falling edge of "TP_USTAW_DELAY_SIŁ_ZAG"
   "m_zboczeN_ustaw_delay_zagn" := "TP_USTAW_DELAY_SIŁ_ZAG";
   IF #_w4 THEN "proces_value".db_tp_nowy_delay_sił_zag := 0.0; END_IF;
   #_w5 := "AlwaysTRUE" AND NOT "TP_USTAW_DELAY_SIŁ_ODB" AND "m_zboczeN_ustaw_delay_odbioru";   // falling edge of "TP_USTAW_DELAY_SIŁ_ODB"
   "m_zboczeN_ustaw_delay_odbioru" := "TP_USTAW_DELAY_SIŁ_ODB";
   IF #_w5 THEN "proces_value".db_tp_nowy_delay_sił_odbioru_stoł := 0.0; END_IF;
END_REGION
END_FUNCTION

FUNCTION "SERVO" : Void   // FC4, LAD
{ S7_Optimized_Access := 'TRUE' }
VERSION : 0.1
// stored: AutoNumber true, IsIECCheckEnabled false, SetENOAutomatically false, UDAEnableTagReadback false
   VAR_TEMP
      Actual_position : Real;
   END_VAR
   VAR_TEMP   // added for the SCL form of the ladder/FBD networks
      _w1 : Bool;
   END_VAR
BEGIN

REGION Network 1: POWER ON
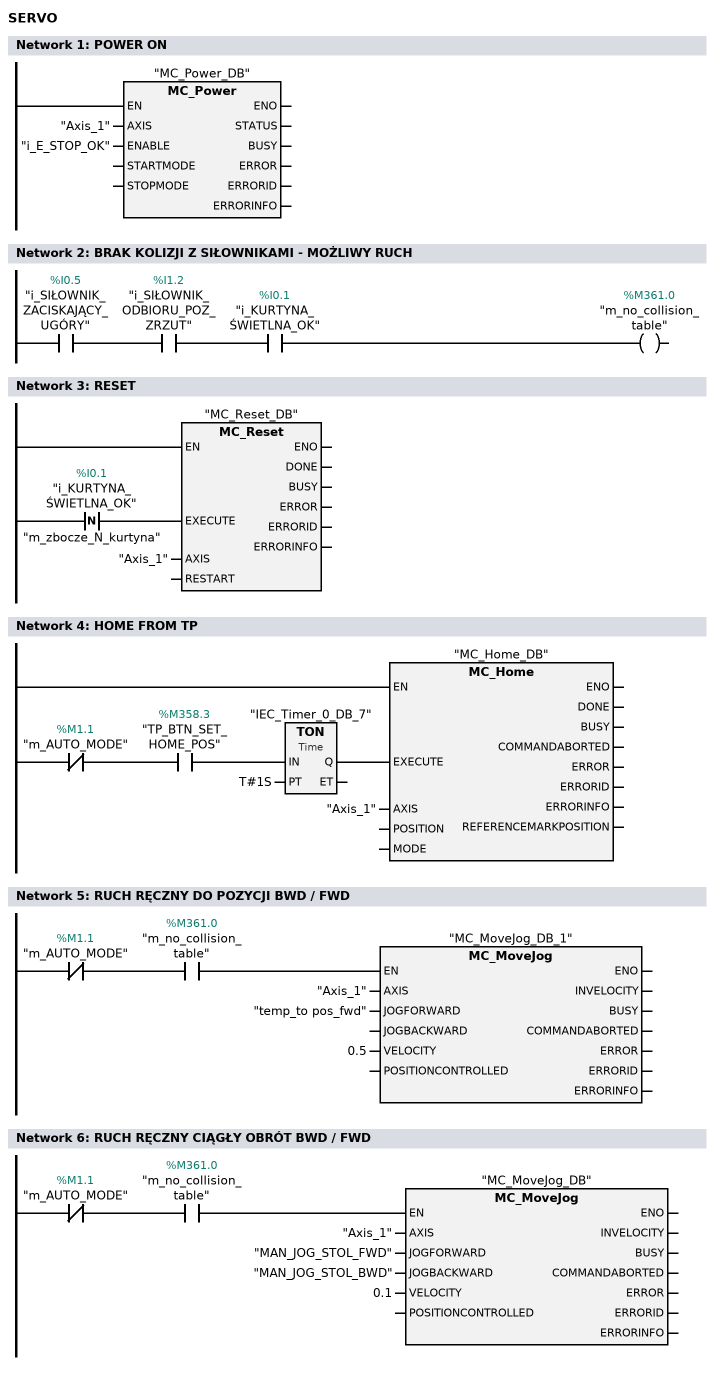
   RUNG wire#powerrail
      "MC_Power_DB".MC_Power(Axis := "Axis_1", Enable := "i_E_STOP_OK", StartMode :=, StopMode :=, Status =>, Busy =>, Error =>, ErrorID =>, ErrorInfo =>)
   END_RUNG
   // the same network as SCL:
   "MC_Power_DB"(Axis := "Axis_1", Enable := "i_E_STOP_OK");   // MC_Power
END_REGION

REGION Network 2: BRAK KOLIZJI Z SIŁOWNIKAMI - MOŻLIWY RUCH
   RUNG wire#powerrail
      Contact( "i_SIŁOWNIK_ZACISKAJĄCY_UGÓRY" )
      Contact( "i_SIŁOWNIK_ODBIORU_POZ_ZRZUT" )
      Contact( "i_KURTYNA_ŚWIETLNA_OK" )
      Coil( "m_no_collision_table" )
   END_RUNG
   // the same network as SCL:
   "m_no_collision_table" := "i_SIŁOWNIK_ZACISKAJĄCY_UGÓRY" AND "i_SIŁOWNIK_ODBIORU_POZ_ZRZUT" AND "i_KURTYNA_ŚWIETLNA_OK";
END_REGION

REGION Network 3: RESET
   RUNG wire#powerrail
      "MC_Reset_DB".MC_Reset(Execute := wire#w1, Axis := "Axis_1", Restart :=, Done =>, Busy =>, Error =>, ErrorID =>, ErrorInfo =>)
   END_RUNG
   RUNG wire#powerrail
      N_Contact(operand := "i_KURTYNA_ŚWIETLNA_OK", bit := "m_zbocze_N_kurtyna")
   END_RUNG wire#w1
   // the same network as SCL:
   #_w1 := NOT "i_KURTYNA_ŚWIETLNA_OK" AND "m_zbocze_N_kurtyna";   // falling edge of "i_KURTYNA_ŚWIETLNA_OK"
   "m_zbocze_N_kurtyna" := "i_KURTYNA_ŚWIETLNA_OK";
   "MC_Reset_DB"(Execute := #_w1, Axis := "Axis_1");   // MC_Reset
END_REGION

REGION Network 4: HOME FROM TP
   RUNG wire#powerrail
      "MC_Home_DB".MC_Home(Execute := wire#w1, Axis := "Axis_1", Position :=, Mode :=, Done =>, Busy =>, CommandAborted =>, Error =>, ErrorID =>, ErrorInfo =>, ReferenceMarkPosition =>)
   END_RUNG
   RUNG wire#powerrail
      I_Contact( "m_AUTO_MODE" )
      Contact( "TP_BTN_SET_HOME_POS" )
      { S7_Templates := "time_type := Time" } "IEC_Timer_0_DB_7".TON(pt := T#1S, et =>)
   END_RUNG wire#w1
   // the same network as SCL:
   "IEC_Timer_0_DB_7".TON(IN := NOT "m_AUTO_MODE" AND "TP_BTN_SET_HOME_POS", PT := T#1S);
   "MC_Home_DB"(Execute := "IEC_Timer_0_DB_7".Q, Axis := "Axis_1");   // MC_Home
END_REGION

REGION Network 5: RUCH RĘCZNY DO POZYCJI BWD / FWD
   RUNG wire#powerrail
      I_Contact( "m_AUTO_MODE" )
      Contact( "m_no_collision_table" )
      "MC_MoveJog_DB_1".MC_MoveJog(Axis := "Axis_1", JogForward := "temp_to pos_fwd", JogBackward :=, Velocity := 0.5, PositionControlled :=, InVelocity =>, Busy =>, CommandAborted =>, Error =>, ErrorID =>, ErrorInfo =>)
   END_RUNG
   // the same network as SCL:
   IF NOT "m_AUTO_MODE" AND "m_no_collision_table" THEN
       "MC_MoveJog_DB_1"(Axis := "Axis_1", JogForward := "temp_to pos_fwd", Velocity := 0.5);   // MC_MoveJog
   END_IF;
END_REGION

REGION Network 6: RUCH RĘCZNY CIĄGŁY OBRÓT BWD / FWD
   RUNG wire#powerrail
      I_Contact( "m_AUTO_MODE" )
      Contact( "m_no_collision_table" )
      "MC_MoveJog_DB".MC_MoveJog(Axis := "Axis_1", JogForward := "MAN_JOG_STOL_FWD", JogBackward := "MAN_JOG_STOL_BWD", Velocity := 0.1, PositionControlled :=, InVelocity =>, Busy =>, CommandAborted =>, Error =>, ErrorID =>, ErrorInfo =>)
   END_RUNG
   // the same network as SCL:
   IF NOT "m_AUTO_MODE" AND "m_no_collision_table" THEN
       "MC_MoveJog_DB"(Axis := "Axis_1",   // MC_MoveJog
                       JogForward := "MAN_JOG_STOL_FWD",
                       JogBackward := "MAN_JOG_STOL_BWD",
                       Velocity := 0.1);
   END_IF;
END_REGION
END_FUNCTION

FUNCTION "AUTOMAT" : Void   // FC6, LAD
{ S7_Optimized_Access := 'TRUE' }
VERSION : 0.1
// stored: AutoNumber true, IsIECCheckEnabled false, SetENOAutomatically false, UDAEnableTagReadback false
   VAR_TEMP
      m_zbocze_czujnik_poz_odb_stoł : Bool;
      m_zbocze_czujnik_stołP : Bool;
      m_zboczeN_czuj_plyt_przód : Bool;
      m_memo_stol_poz : Bool;
   END_VAR
   VAR_TEMP   // added for the SCL form of the ladder/FBD networks
      _w1 : Bool;
      _w2 : Bool;
   END_VAR
BEGIN

REGION Network 1: CHECK SERVO CONDITIONS
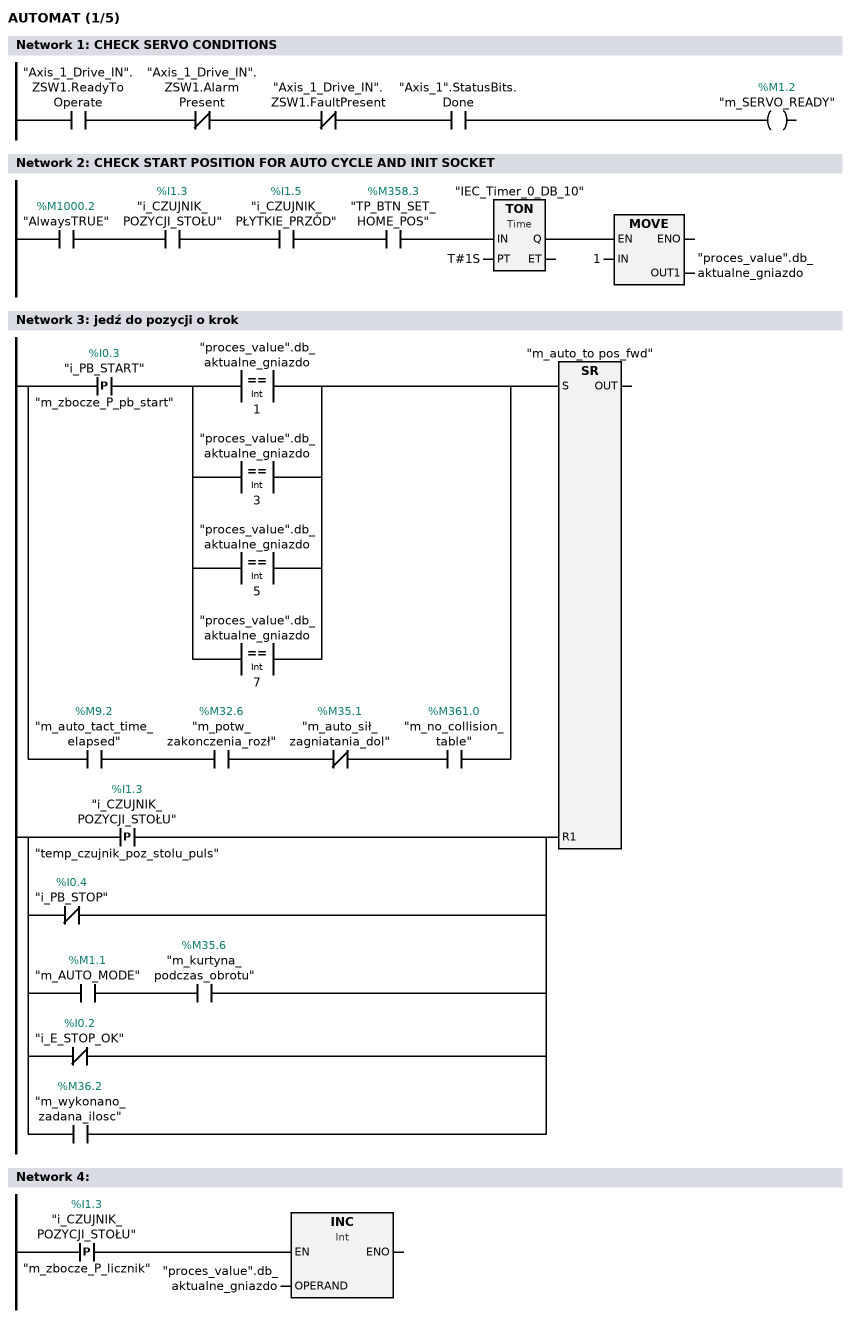
   RUNG wire#powerrail
      Contact( "Axis_1_Drive_IN".ZSW1.ReadyToOperate )
      I_Contact( "Axis_1_Drive_IN".ZSW1.AlarmPresent )
      I_Contact( "Axis_1_Drive_IN".ZSW1.FaultPresent )
      Contact( "Axis_1".StatusBits.Done )
      Coil( "m_SERVO_READY" )
   END_RUNG
   // the same network as SCL:
   "m_SERVO_READY" := "Axis_1_Drive_IN".ZSW1.ReadyToOperate AND NOT "Axis_1_Drive_IN".ZSW1.AlarmPresent AND NOT "Axis_1_Drive_IN".ZSW1.FaultPresent AND "Axis_1".StatusBits.Done;
END_REGION

REGION Network 2: CHECK START POSITION FOR AUTO CYCLE AND INIT SOCKET
   RUNG wire#powerrail
      Contact( "AlwaysTRUE" )
      Contact( "i_CZUJNIK_POZYCJI_STOŁU" )
      Contact( "i_CZUJNIK_PŁYTKIE_PRZÓD" )
      Contact( "TP_BTN_SET_HOME_POS" )
      { S7_Templates := "time_type := Time" } "IEC_Timer_0_DB_10".TON(pt := T#1S, et =>)
      Move(in := 1, out1 => "proces_value".db_aktualne_gniazdo)
   END_RUNG
   // the same network as SCL:
   "IEC_Timer_0_DB_10".TON(IN := "AlwaysTRUE" AND "i_CZUJNIK_POZYCJI_STOŁU" AND "i_CZUJNIK_PŁYTKIE_PRZÓD" AND "TP_BTN_SET_HOME_POS",
                           PT := T#1S);
   IF "IEC_Timer_0_DB_10".Q THEN "proces_value".db_aktualne_gniazdo := 1; END_IF;
END_REGION

REGION Network 3: jedź do pozycji o krok
   RUNG wire#powerrail
      P_Contact(operand := "i_PB_START", bit := "m_zbocze_P_pb_start")
      wire#w1
      { S7_Templates := "SrcType := Int" } EQ_Contact(in1 := "proces_value".db_aktualne_gniazdo, in2 := 1)
      wire#w2
      S_SR(operand := "m_auto_to pos_fwd", r1 := wire#w3)
   END_RUNG
   RUNG wire#w1
      { S7_Templates := "SrcType := Int" } EQ_Contact(in1 := "proces_value".db_aktualne_gniazdo, in2 := 3)
   END_RUNG wire#w2
   RUNG wire#w1
      { S7_Templates := "SrcType := Int" } EQ_Contact(in1 := "proces_value".db_aktualne_gniazdo, in2 := 5)
   END_RUNG wire#w2
   RUNG wire#w1
      { S7_Templates := "SrcType := Int" } EQ_Contact(in1 := "proces_value".db_aktualne_gniazdo, in2 := 7)
   END_RUNG wire#w2
   RUNG wire#powerrail
      Contact( "m_auto_tact_time_elapsed" )
      Contact( "m_potw_zakonczenia_rozł" )
      I_Contact( "m_auto_sił_zagniatania_dol" )
      Contact( "m_no_collision_table" )
   END_RUNG wire#w2
   RUNG wire#powerrail
      P_Contact(operand := "i_CZUJNIK_POZYCJI_STOŁU", bit := "temp_czujnik_poz_stolu_puls")
   END_RUNG wire#w3
   RUNG wire#powerrail
      I_Contact( "i_PB_STOP" )
   END_RUNG wire#w3
   RUNG wire#powerrail
      Contact( "m_AUTO_MODE" )
      Contact( "m_kurtyna_podczas_obrotu" )
   END_RUNG wire#w3
   RUNG wire#powerrail
      I_Contact( "i_E_STOP_OK" )
   END_RUNG wire#w3
   RUNG wire#powerrail
      Contact( "m_wykonano_zadana_ilosc" )
   END_RUNG wire#w3
   // the same network as SCL:
   #_w1 := "i_PB_START" AND NOT "m_zbocze_P_pb_start";   // rising edge of "i_PB_START"
   "m_zbocze_P_pb_start" := "i_PB_START";
   #_w2 := "i_CZUJNIK_POZYCJI_STOŁU" AND NOT "temp_czujnik_poz_stolu_puls";   // rising edge of "i_CZUJNIK_POZYCJI_STOŁU"
   "temp_czujnik_poz_stolu_puls" := "i_CZUJNIK_POZYCJI_STOŁU";
   IF (#_w1 AND (("proces_value".db_aktualne_gniazdo = 1) OR ("proces_value".db_aktualne_gniazdo = 3) OR ("proces_value".db_aktualne_gniazdo = 5) OR ("proces_value".db_aktualne_gniazdo = 7))) OR ("m_auto_tact_time_elapsed" AND "m_potw_zakonczenia_rozł" AND NOT "m_auto_sił_zagniatania_dol" AND "m_no_collision_table") THEN
       "m_auto_to pos_fwd" := TRUE;   // SR flip-flop
   END_IF;
   IF #_w2 OR NOT "i_PB_STOP" OR ("m_AUTO_MODE" AND "m_kurtyna_podczas_obrotu") OR NOT "i_E_STOP_OK" OR "m_wykonano_zadana_ilosc" THEN
       "m_auto_to pos_fwd" := FALSE;
   END_IF;
END_REGION

REGION Network 4
   RUNG wire#powerrail
      P_Contact(operand := "i_CZUJNIK_POZYCJI_STOŁU", bit := "m_zbocze_P_licznik")
      { S7_Templates := "DestType := Int" } Inc( "proces_value".db_aktualne_gniazdo )
   END_RUNG
   // the same network as SCL:
   #_w1 := "i_CZUJNIK_POZYCJI_STOŁU" AND NOT "m_zbocze_P_licznik";   // rising edge of "i_CZUJNIK_POZYCJI_STOŁU"
   "m_zbocze_P_licznik" := "i_CZUJNIK_POZYCJI_STOŁU";
   IF #_w1 THEN "proces_value".db_aktualne_gniazdo := "proces_value".db_aktualne_gniazdo + 1; END_IF;
END_REGION

REGION Network 5
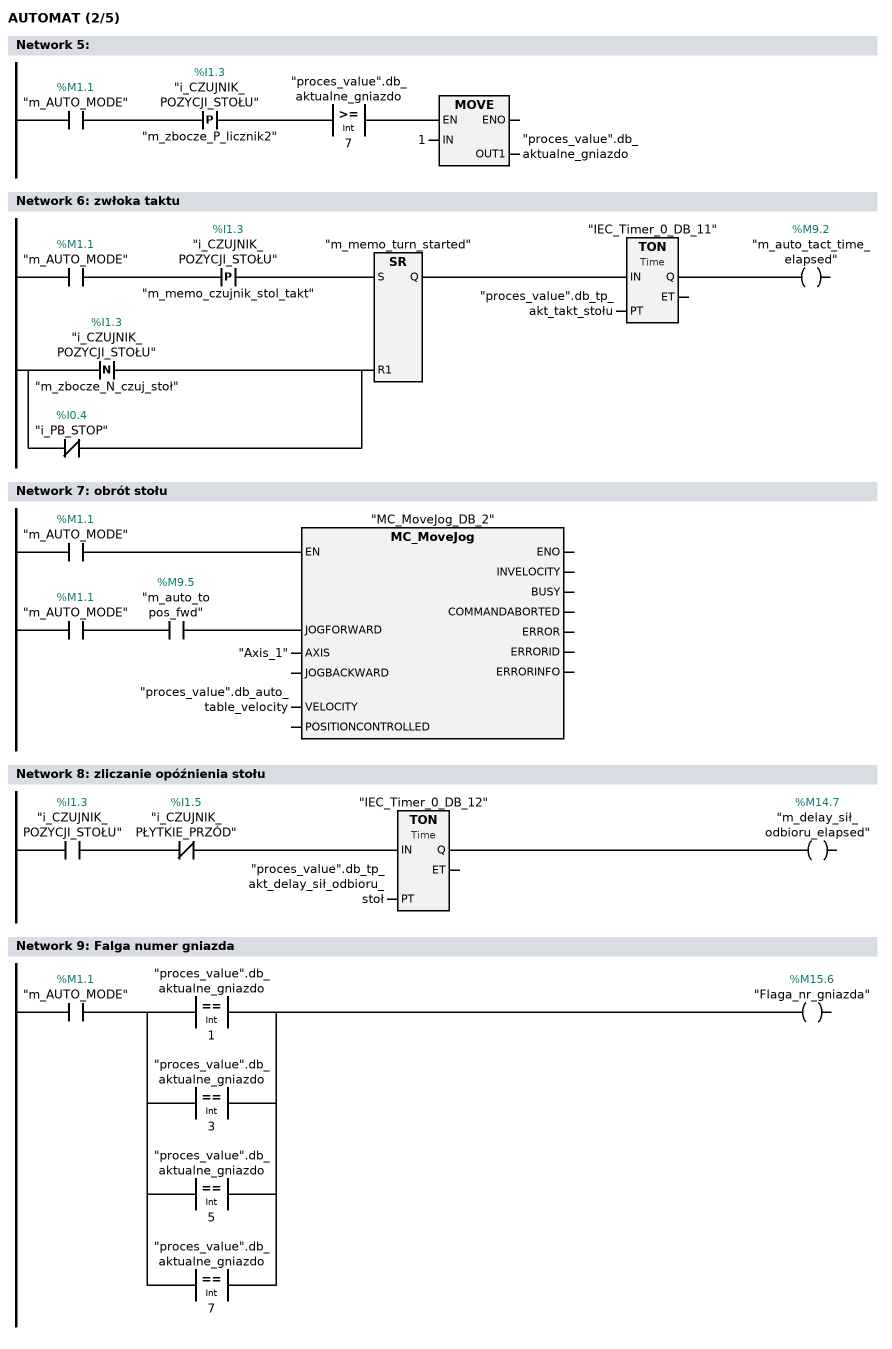
   RUNG wire#powerrail
      Contact( "m_AUTO_MODE" )
      P_Contact(operand := "i_CZUJNIK_POZYCJI_STOŁU", bit := "m_zbocze_P_licznik2")
      { S7_Templates := "SrcType := Int" } GE_Contact(in1 := "proces_value".db_aktualne_gniazdo, in2 := 7)
      Move(in := 1, out1 => "proces_value".db_aktualne_gniazdo)
   END_RUNG
   // the same network as SCL:
   #_w1 := "m_AUTO_MODE" AND "i_CZUJNIK_POZYCJI_STOŁU" AND NOT "m_zbocze_P_licznik2";   // rising edge of "i_CZUJNIK_POZYCJI_STOŁU"
   "m_zbocze_P_licznik2" := "i_CZUJNIK_POZYCJI_STOŁU";
   IF #_w1 AND ("proces_value".db_aktualne_gniazdo >= 7) THEN
       "proces_value".db_aktualne_gniazdo := 1;
   END_IF;
END_REGION

REGION Network 6: zwłoka taktu
   RUNG wire#powerrail
      Contact( "m_AUTO_MODE" )
      P_Contact(operand := "i_CZUJNIK_POZYCJI_STOŁU", bit := "m_memo_czujnik_stol_takt")
      S_SR(operand := "m_memo_turn_started", r1 := wire#w1)
      { S7_Templates := "time_type := Time" } "IEC_Timer_0_DB_11".TON(pt := "proces_value".db_tp_akt_takt_stołu, et =>)
      Coil( "m_auto_tact_time_elapsed" )
   END_RUNG
   RUNG wire#powerrail
      N_Contact(operand := "i_CZUJNIK_POZYCJI_STOŁU", bit := "m_zbocze_N_czuj_stoł")
   END_RUNG wire#w1
   RUNG wire#powerrail
      I_Contact( "i_PB_STOP" )
   END_RUNG wire#w1
   // the same network as SCL:
   #_w1 := "m_AUTO_MODE" AND "i_CZUJNIK_POZYCJI_STOŁU" AND NOT "m_memo_czujnik_stol_takt";   // rising edge of "i_CZUJNIK_POZYCJI_STOŁU"
   "m_memo_czujnik_stol_takt" := "i_CZUJNIK_POZYCJI_STOŁU";
   #_w2 := NOT "i_CZUJNIK_POZYCJI_STOŁU" AND "m_zbocze_N_czuj_stoł";   // falling edge of "i_CZUJNIK_POZYCJI_STOŁU"
   "m_zbocze_N_czuj_stoł" := "i_CZUJNIK_POZYCJI_STOŁU";
   IF #_w1 THEN
       "m_memo_turn_started" := TRUE;   // SR flip-flop
   END_IF;
   IF #_w2 OR NOT "i_PB_STOP" THEN "m_memo_turn_started" := FALSE; END_IF;
   "IEC_Timer_0_DB_11".TON(IN := "m_memo_turn_started", PT := "proces_value".db_tp_akt_takt_stołu);
   "m_auto_tact_time_elapsed" := "IEC_Timer_0_DB_11".Q;
END_REGION

REGION Network 7: obrót stołu
   RUNG wire#powerrail
      Contact( "m_AUTO_MODE" )
      "MC_MoveJog_DB_2".MC_MoveJog(JogForward := wire#w1, Axis := "Axis_1", JogBackward :=, Velocity := "proces_value".db_auto_table_velocity, PositionControlled :=, InVelocity =>, Busy =>, CommandAborted =>, Error =>, ErrorID =>, ErrorInfo =>)
   END_RUNG
   RUNG wire#powerrail
      Contact( "m_AUTO_MODE" )
      Contact( "m_auto_to pos_fwd" )
   END_RUNG wire#w1
   // the same network as SCL:
   IF "m_AUTO_MODE" THEN
       "MC_MoveJog_DB_2"(JogForward := "m_AUTO_MODE" AND "m_auto_to pos_fwd",   // MC_MoveJog
                         Axis := "Axis_1",
                         Velocity := "proces_value".db_auto_table_velocity);
   END_IF;
END_REGION

REGION Network 8: zliczanie opóźnienia stołu
   RUNG wire#powerrail
      Contact( "i_CZUJNIK_POZYCJI_STOŁU" )
      I_Contact( "i_CZUJNIK_PŁYTKIE_PRZÓD" )
      { S7_Templates := "time_type := Time" } "IEC_Timer_0_DB_12".TON(pt := "proces_value".db_tp_akt_delay_sił_odbioru_stoł, et =>)
      Coil( "m_delay_sił_odbioru_elapsed" )
   END_RUNG
   // the same network as SCL:
   "IEC_Timer_0_DB_12".TON(IN := "i_CZUJNIK_POZYCJI_STOŁU" AND NOT "i_CZUJNIK_PŁYTKIE_PRZÓD",
                           PT := "proces_value".db_tp_akt_delay_sił_odbioru_stoł);
   "m_delay_sił_odbioru_elapsed" := "IEC_Timer_0_DB_12".Q;
END_REGION

REGION Network 9: Falga numer gniazda
   RUNG wire#powerrail
      Contact( "m_AUTO_MODE" )
      wire#w1
      { S7_Templates := "SrcType := Int" } EQ_Contact(in1 := "proces_value".db_aktualne_gniazdo, in2 := 1)
      wire#w2
      Coil( "Flaga_nr_gniazda" )
   END_RUNG
   RUNG wire#w1
      { S7_Templates := "SrcType := Int" } EQ_Contact(in1 := "proces_value".db_aktualne_gniazdo, in2 := 3)
   END_RUNG wire#w2
   RUNG wire#w1
      { S7_Templates := "SrcType := Int" } EQ_Contact(in1 := "proces_value".db_aktualne_gniazdo, in2 := 5)
   END_RUNG wire#w2
   RUNG wire#w1
      { S7_Templates := "SrcType := Int" } EQ_Contact(in1 := "proces_value".db_aktualne_gniazdo, in2 := 7)
   END_RUNG wire#w2
   // the same network as SCL:
   "Flaga_nr_gniazda" := "m_AUTO_MODE" AND (("proces_value".db_aktualne_gniazdo = 1) OR ("proces_value".db_aktualne_gniazdo = 3) OR ("proces_value".db_aktualne_gniazdo = 5) OR ("proces_value".db_aktualne_gniazdo = 7));
END_REGION

REGION Network 10: siłownik odbioru
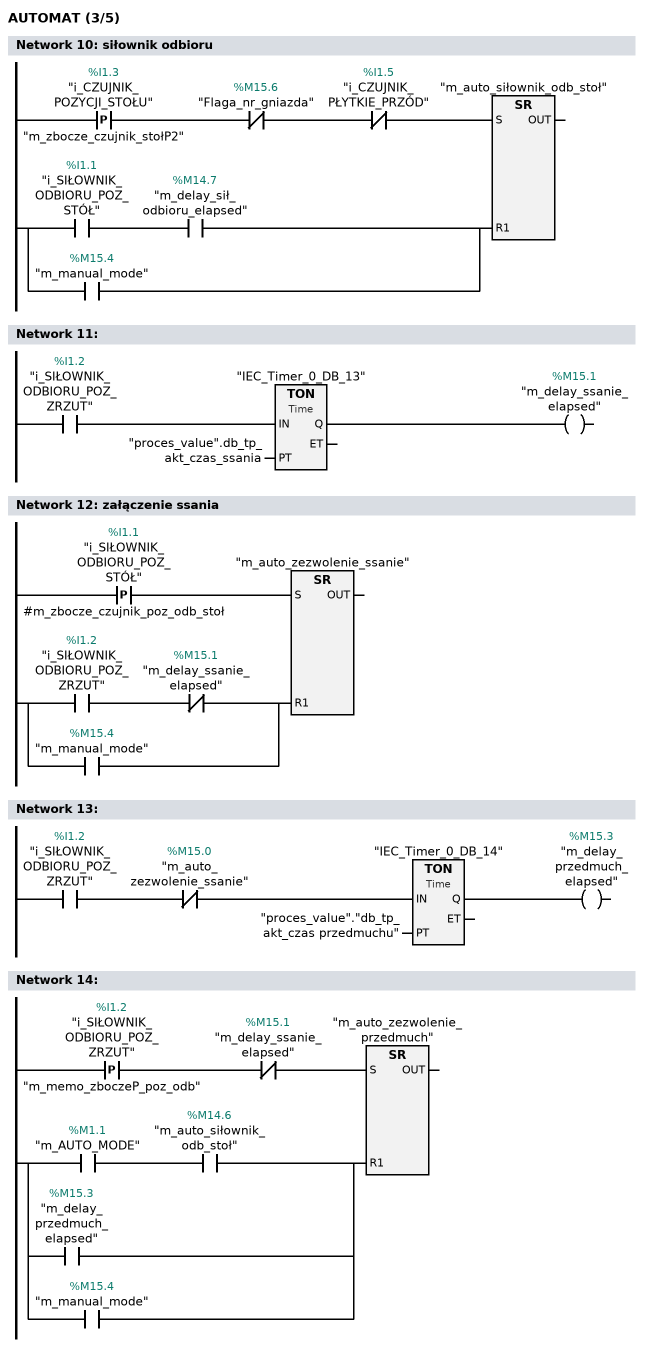
   RUNG wire#powerrail
      P_Contact(operand := "i_CZUJNIK_POZYCJI_STOŁU", bit := "m_zbocze_czujnik_stołP2")
      I_Contact( "Flaga_nr_gniazda" )
      I_Contact( "i_CZUJNIK_PŁYTKIE_PRZÓD" )
      S_SR(operand := "m_auto_siłownik_odb_stoł", r1 := wire#w1)
   END_RUNG
   RUNG wire#powerrail
      Contact( "i_SIŁOWNIK_ODBIORU_POZ_STÓŁ" )
      Contact( "m_delay_sił_odbioru_elapsed" )
   END_RUNG wire#w1
   RUNG wire#powerrail
      Contact( "m_manual_mode" )
   END_RUNG wire#w1
   // the same network as SCL:
   #_w1 := "i_CZUJNIK_POZYCJI_STOŁU" AND NOT "m_zbocze_czujnik_stołP2";   // rising edge of "i_CZUJNIK_POZYCJI_STOŁU"
   "m_zbocze_czujnik_stołP2" := "i_CZUJNIK_POZYCJI_STOŁU";
   IF #_w1 AND NOT "Flaga_nr_gniazda" AND NOT "i_CZUJNIK_PŁYTKIE_PRZÓD" THEN
       "m_auto_siłownik_odb_stoł" := TRUE;   // SR flip-flop
   END_IF;
   IF ("i_SIŁOWNIK_ODBIORU_POZ_STÓŁ" AND "m_delay_sił_odbioru_elapsed") OR "m_manual_mode" THEN
       "m_auto_siłownik_odb_stoł" := FALSE;
   END_IF;
END_REGION

REGION Network 11
   RUNG wire#powerrail
      Contact( "i_SIŁOWNIK_ODBIORU_POZ_ZRZUT" )
      { S7_Templates := "time_type := Time" } "IEC_Timer_0_DB_13".TON(pt := "proces_value".db_tp_akt_czas_ssania, et =>)
      Coil( "m_delay_ssanie_elapsed" )
   END_RUNG
   // the same network as SCL:
   "IEC_Timer_0_DB_13".TON(IN := "i_SIŁOWNIK_ODBIORU_POZ_ZRZUT", PT := "proces_value".db_tp_akt_czas_ssania);
   "m_delay_ssanie_elapsed" := "IEC_Timer_0_DB_13".Q;
END_REGION

REGION Network 12: załączenie ssania
   RUNG wire#powerrail
      P_Contact(operand := "i_SIŁOWNIK_ODBIORU_POZ_STÓŁ", bit := #m_zbocze_czujnik_poz_odb_stoł)
      S_SR(operand := "m_auto_zezwolenie_ssanie", r1 := wire#w1)
   END_RUNG
   RUNG wire#powerrail
      Contact( "i_SIŁOWNIK_ODBIORU_POZ_ZRZUT" )
      I_Contact( "m_delay_ssanie_elapsed" )
   END_RUNG wire#w1
   RUNG wire#powerrail
      Contact( "m_manual_mode" )
   END_RUNG wire#w1
   // the same network as SCL:
   #_w1 := "i_SIŁOWNIK_ODBIORU_POZ_STÓŁ" AND NOT #m_zbocze_czujnik_poz_odb_stoł;   // rising edge of "i_SIŁOWNIK_ODBIORU_POZ_STÓŁ"
   #m_zbocze_czujnik_poz_odb_stoł := "i_SIŁOWNIK_ODBIORU_POZ_STÓŁ";
   IF #_w1 THEN
       "m_auto_zezwolenie_ssanie" := TRUE;   // SR flip-flop
   END_IF;
   IF ("i_SIŁOWNIK_ODBIORU_POZ_ZRZUT" AND NOT "m_delay_ssanie_elapsed") OR "m_manual_mode" THEN
       "m_auto_zezwolenie_ssanie" := FALSE;
   END_IF;
END_REGION

REGION Network 13
   RUNG wire#powerrail
      Contact( "i_SIŁOWNIK_ODBIORU_POZ_ZRZUT" )
      I_Contact( "m_auto_zezwolenie_ssanie" )
      { S7_Templates := "time_type := Time" } "IEC_Timer_0_DB_14".TON(pt := "proces_value"."db_tp_akt_czas przedmuchu", et =>)
      Coil( "m_delay_przedmuch_elapsed" )
   END_RUNG
   // the same network as SCL:
   "IEC_Timer_0_DB_14".TON(IN := "i_SIŁOWNIK_ODBIORU_POZ_ZRZUT" AND NOT "m_auto_zezwolenie_ssanie",
                           PT := "proces_value"."db_tp_akt_czas przedmuchu");
   "m_delay_przedmuch_elapsed" := "IEC_Timer_0_DB_14".Q;
END_REGION

REGION Network 14
   RUNG wire#powerrail
      P_Contact(operand := "i_SIŁOWNIK_ODBIORU_POZ_ZRZUT", bit := "m_memo_zboczeP_poz_odb")
      I_Contact( "m_delay_ssanie_elapsed" )
      S_SR(operand := "m_auto_zezwolenie_przedmuch", r1 := wire#w1)
   END_RUNG
   RUNG wire#powerrail
      Contact( "m_AUTO_MODE" )
      Contact( "m_auto_siłownik_odb_stoł" )
   END_RUNG wire#w1
   RUNG wire#powerrail
      Contact( "m_delay_przedmuch_elapsed" )
   END_RUNG wire#w1
   RUNG wire#powerrail
      Contact( "m_manual_mode" )
   END_RUNG wire#w1
   // the same network as SCL:
   #_w1 := "i_SIŁOWNIK_ODBIORU_POZ_ZRZUT" AND NOT "m_memo_zboczeP_poz_odb";   // rising edge of "i_SIŁOWNIK_ODBIORU_POZ_ZRZUT"
   "m_memo_zboczeP_poz_odb" := "i_SIŁOWNIK_ODBIORU_POZ_ZRZUT";
   IF #_w1 AND NOT "m_delay_ssanie_elapsed" THEN
       "m_auto_zezwolenie_przedmuch" := TRUE;   // SR flip-flop
   END_IF;
   IF ("m_AUTO_MODE" AND "m_auto_siłownik_odb_stoł") OR "m_delay_przedmuch_elapsed" OR "m_manual_mode" THEN
       "m_auto_zezwolenie_przedmuch" := FALSE;
   END_IF;
END_REGION

REGION Network 15: rozładunek zakończony
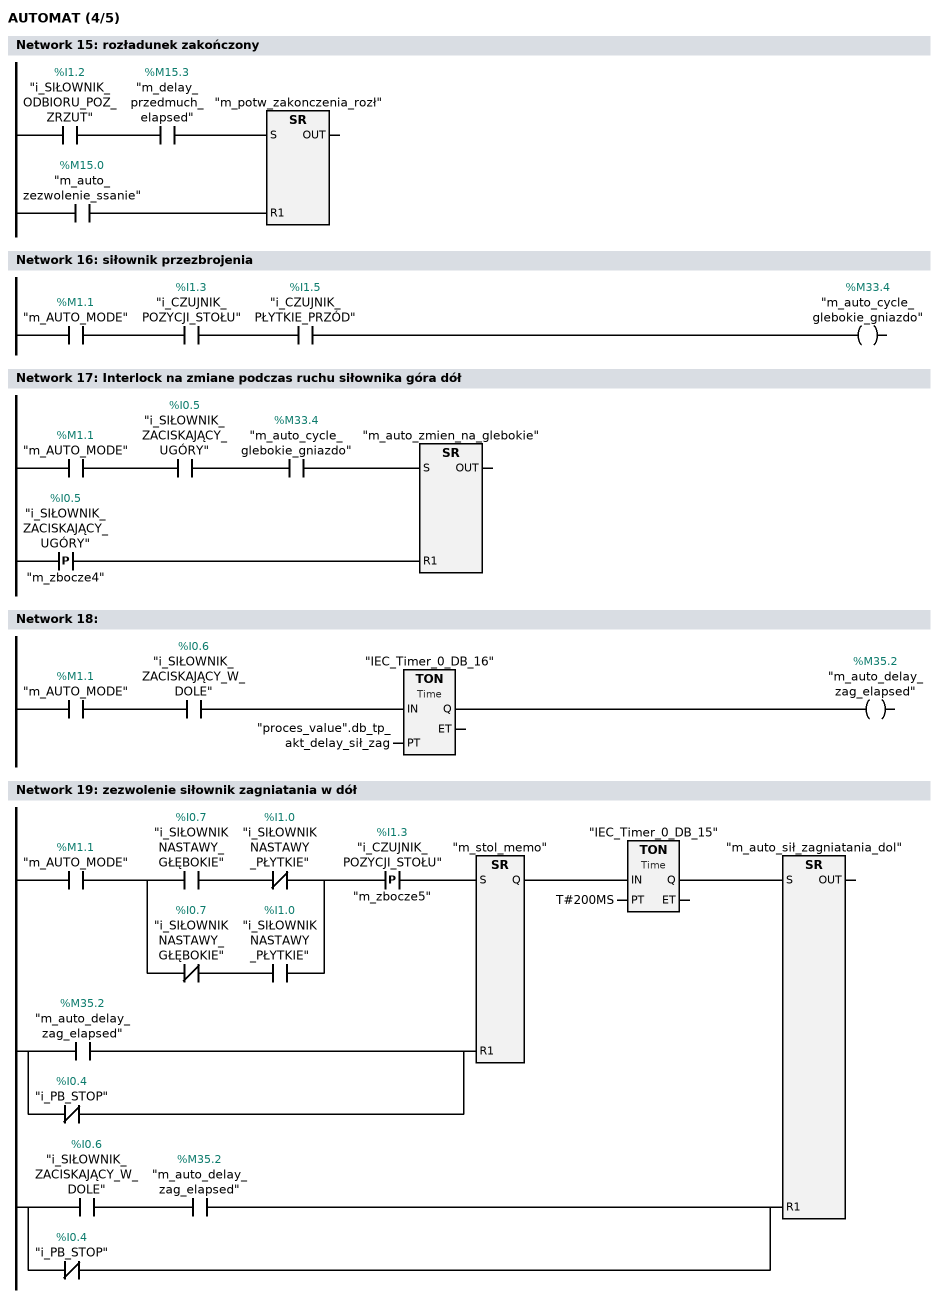
   RUNG wire#powerrail
      Contact( "i_SIŁOWNIK_ODBIORU_POZ_ZRZUT" )
      Contact( "m_delay_przedmuch_elapsed" )
      S_SR(operand := "m_potw_zakonczenia_rozł", r1 := wire#w1)
   END_RUNG
   RUNG wire#powerrail
      Contact( "m_auto_zezwolenie_ssanie" )
   END_RUNG wire#w1
   // the same network as SCL:
   IF "i_SIŁOWNIK_ODBIORU_POZ_ZRZUT" AND "m_delay_przedmuch_elapsed" THEN
       "m_potw_zakonczenia_rozł" := TRUE;   // SR flip-flop
   END_IF;
   IF "m_auto_zezwolenie_ssanie" THEN "m_potw_zakonczenia_rozł" := FALSE; END_IF;
END_REGION

REGION Network 16: siłownik przezbrojenia
   RUNG wire#powerrail
      Contact( "m_AUTO_MODE" )
      Contact( "i_CZUJNIK_POZYCJI_STOŁU" )
      Contact( "i_CZUJNIK_PŁYTKIE_PRZÓD" )
      Coil( "m_auto_cycle_glebokie_gniazdo" )
   END_RUNG
   // the same network as SCL:
   "m_auto_cycle_glebokie_gniazdo" := "m_AUTO_MODE" AND "i_CZUJNIK_POZYCJI_STOŁU" AND "i_CZUJNIK_PŁYTKIE_PRZÓD";
END_REGION

REGION Network 17: Interlock na zmiane podczas ruchu siłownika góra dół
   RUNG wire#powerrail
      Contact( "m_AUTO_MODE" )
      Contact( "i_SIŁOWNIK_ZACISKAJĄCY_UGÓRY" )
      Contact( "m_auto_cycle_glebokie_gniazdo" )
      S_SR(operand := "m_auto_zmien_na_glebokie", r1 := wire#w1)
   END_RUNG
   RUNG wire#powerrail
      P_Contact(operand := "i_SIŁOWNIK_ZACISKAJĄCY_UGÓRY", bit := "m_zbocze4")
   END_RUNG wire#w1
   // the same network as SCL:
   #_w1 := "i_SIŁOWNIK_ZACISKAJĄCY_UGÓRY" AND NOT "m_zbocze4";   // rising edge of "i_SIŁOWNIK_ZACISKAJĄCY_UGÓRY"
   "m_zbocze4" := "i_SIŁOWNIK_ZACISKAJĄCY_UGÓRY";
   IF "m_AUTO_MODE" AND "i_SIŁOWNIK_ZACISKAJĄCY_UGÓRY" AND "m_auto_cycle_glebokie_gniazdo" THEN
       "m_auto_zmien_na_glebokie" := TRUE;   // SR flip-flop
   END_IF;
   IF #_w1 THEN "m_auto_zmien_na_glebokie" := FALSE; END_IF;
END_REGION

REGION Network 18
   RUNG wire#powerrail
      Contact( "m_AUTO_MODE" )
      Contact( "i_SIŁOWNIK_ZACISKAJĄCY_W_DOLE" )
      { S7_Templates := "time_type := Time" } "IEC_Timer_0_DB_16".TON(pt := "proces_value".db_tp_akt_delay_sił_zag, et =>)
      Coil( "m_auto_delay_zag_elapsed" )
   END_RUNG
   // the same network as SCL:
   "IEC_Timer_0_DB_16".TON(IN := "m_AUTO_MODE" AND "i_SIŁOWNIK_ZACISKAJĄCY_W_DOLE",
                           PT := "proces_value".db_tp_akt_delay_sił_zag);
   "m_auto_delay_zag_elapsed" := "IEC_Timer_0_DB_16".Q;
END_REGION

REGION Network 19: zezwolenie siłownik zagniatania w dół
   RUNG wire#powerrail
      Contact( "m_AUTO_MODE" )
      wire#w1
      Contact( "i_SIŁOWNIK NASTAWY_GŁĘBOKIE" )
      I_Contact( "i_SIŁOWNIK NASTAWY _PŁYTKIE" )
      wire#w2
      P_Contact(operand := "i_CZUJNIK_POZYCJI_STOŁU", bit := "m_zbocze5")
      S_SR(operand := "m_stol_memo", r1 := wire#w3)
      { S7_Templates := "time_type := Time" } "IEC_Timer_0_DB_15".TON(pt := T#200MS, et =>)
      S_SR(operand := "m_auto_sił_zagniatania_dol", r1 := wire#w4)
   END_RUNG
   RUNG wire#w1
      I_Contact( "i_SIŁOWNIK NASTAWY_GŁĘBOKIE" )
      Contact( "i_SIŁOWNIK NASTAWY _PŁYTKIE" )
   END_RUNG wire#w2
   RUNG wire#powerrail
      Contact( "m_auto_delay_zag_elapsed" )
   END_RUNG wire#w3
   RUNG wire#powerrail
      I_Contact( "i_PB_STOP" )
   END_RUNG wire#w3
   RUNG wire#powerrail
      Contact( "i_SIŁOWNIK_ZACISKAJĄCY_W_DOLE" )
      Contact( "m_auto_delay_zag_elapsed" )
   END_RUNG wire#w4
   RUNG wire#powerrail
      I_Contact( "i_PB_STOP" )
   END_RUNG wire#w4
   // the same network as SCL:
   #_w1 := "m_AUTO_MODE" AND (("i_SIŁOWNIK NASTAWY_GŁĘBOKIE" AND NOT "i_SIŁOWNIK NASTAWY _PŁYTKIE") OR (NOT "i_SIŁOWNIK NASTAWY_GŁĘBOKIE" AND "i_SIŁOWNIK NASTAWY _PŁYTKIE")) AND "i_CZUJNIK_POZYCJI_STOŁU" AND NOT "m_zbocze5";   // rising edge of "i_CZUJNIK_POZYCJI_STOŁU"
   "m_zbocze5" := "i_CZUJNIK_POZYCJI_STOŁU";
   IF #_w1 THEN
       "m_stol_memo" := TRUE;   // SR flip-flop
   END_IF;
   IF "m_auto_delay_zag_elapsed" OR NOT "i_PB_STOP" THEN "m_stol_memo" := FALSE; END_IF;
   "IEC_Timer_0_DB_15".TON(IN := "m_stol_memo", PT := T#200MS);
   IF "IEC_Timer_0_DB_15".Q THEN
       "m_auto_sił_zagniatania_dol" := TRUE;   // SR flip-flop
   END_IF;
   IF ("i_SIŁOWNIK_ZACISKAJĄCY_W_DOLE" AND "m_auto_delay_zag_elapsed") OR NOT "i_PB_STOP" THEN
       "m_auto_sił_zagniatania_dol" := FALSE;
   END_IF;
END_REGION

REGION Network 20: dobezpieczenie wejścia podczas obrotu - reset po bazowaniu gniazda
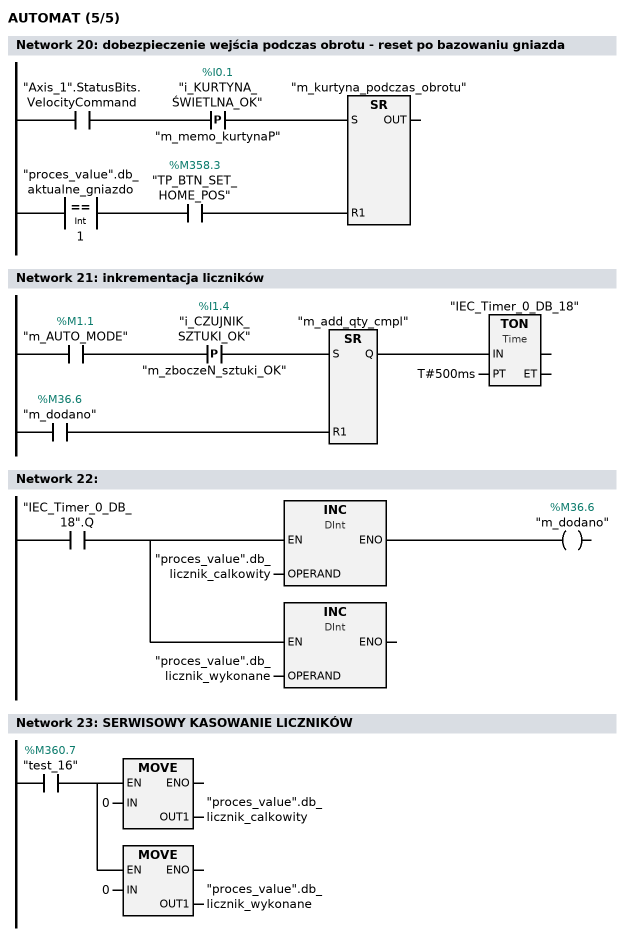
   RUNG wire#powerrail
      Contact( "Axis_1".StatusBits.VelocityCommand )
      P_Contact(operand := "i_KURTYNA_ŚWIETLNA_OK", bit := "m_memo_kurtynaP")
      S_SR(operand := "m_kurtyna_podczas_obrotu", r1 := wire#w1)
   END_RUNG
   RUNG wire#powerrail
      { S7_Templates := "SrcType := Int" } EQ_Contact(in1 := "proces_value".db_aktualne_gniazdo, in2 := 1)
      Contact( "TP_BTN_SET_HOME_POS" )
   END_RUNG wire#w1
   // the same network as SCL:
   #_w1 := "Axis_1".StatusBits.VelocityCommand AND "i_KURTYNA_ŚWIETLNA_OK" AND NOT "m_memo_kurtynaP";   // rising edge of "i_KURTYNA_ŚWIETLNA_OK"
   "m_memo_kurtynaP" := "i_KURTYNA_ŚWIETLNA_OK";
   IF #_w1 THEN
       "m_kurtyna_podczas_obrotu" := TRUE;   // SR flip-flop
   END_IF;
   IF ("proces_value".db_aktualne_gniazdo = 1) AND "TP_BTN_SET_HOME_POS" THEN
       "m_kurtyna_podczas_obrotu" := FALSE;
   END_IF;
END_REGION

REGION Network 21: inkrementacja liczników
   RUNG wire#powerrail
      Contact( "m_AUTO_MODE" )
      P_Contact(operand := "i_CZUJNIK_SZTUKI_OK", bit := "m_zboczeN_sztuki_OK")
      S_SR(operand := "m_add_qty_cmpl", r1 := wire#w1)
      { S7_Templates := "time_type := Time" } "IEC_Timer_0_DB_18".TON(pt := T#500ms, et =>)
   END_RUNG
   RUNG wire#powerrail
      Contact( "m_dodano" )
   END_RUNG wire#w1
   // the same network as SCL:
   #_w1 := "m_AUTO_MODE" AND "i_CZUJNIK_SZTUKI_OK" AND NOT "m_zboczeN_sztuki_OK";   // rising edge of "i_CZUJNIK_SZTUKI_OK"
   "m_zboczeN_sztuki_OK" := "i_CZUJNIK_SZTUKI_OK";
   IF #_w1 THEN
       "m_add_qty_cmpl" := TRUE;   // SR flip-flop
   END_IF;
   IF "m_dodano" THEN "m_add_qty_cmpl" := FALSE; END_IF;
   "IEC_Timer_0_DB_18".TON(IN := "m_add_qty_cmpl", PT := T#500ms);
END_REGION

REGION Network 22
   RUNG wire#powerrail
      Contact( "IEC_Timer_0_DB_18".Q )
      wire#w1
      { S7_Templates := "DestType := DInt" } Inc( "proces_value".db_licznik_calkowity )
      Coil( "m_dodano" )
   END_RUNG
   RUNG wire#w1
      { S7_Templates := "DestType := DInt" } Inc( "proces_value".db_licznik_wykonane )
   END_RUNG
   // the same network as SCL:
   IF "IEC_Timer_0_DB_18".Q THEN
       "proces_value".db_licznik_calkowity := "proces_value".db_licznik_calkowity + 1;
   END_IF;
   "m_dodano" := "IEC_Timer_0_DB_18".Q;
   IF "IEC_Timer_0_DB_18".Q THEN
       "proces_value".db_licznik_wykonane := "proces_value".db_licznik_wykonane + 1;
   END_IF;
END_REGION

REGION Network 23: SERWISOWY KASOWANIE LICZNIKÓW
   RUNG wire#powerrail
      Contact( "test_16" )
      wire#w1
      Move(in := 0, out1 => "proces_value".db_licznik_calkowity)
   END_RUNG
   RUNG wire#w1
      Move(in := 0, out1 => "proces_value".db_licznik_wykonane)
   END_RUNG
   // the same network as SCL:
   IF "test_16" THEN
       "proces_value".db_licznik_calkowity := 0;
       "proces_value".db_licznik_wykonane := 0;
   END_IF;
END_REGION
END_FUNCTION

FUNCTION "INFO" : Void   // FC7, LAD
{ S7_Optimized_Access := 'TRUE' }
VERSION : 0.1
// stored: AutoNumber true, IsIECCheckEnabled false, SetENOAutomatically false, UDAEnableTagReadback false
   VAR_TEMP
      temp_1 : Bool;
      m_temp2 : Bool;
      m_temp3 : Bool;
      m_temp4 : Bool;
      m_puls_liczniki : Bool;
      test1 : Bool;
   END_VAR
   VAR_TEMP   // added for the SCL form of the ladder/FBD networks
      _w1 : Bool;
   END_VAR
BEGIN

REGION Network 1: Powiadomienie o wykonaniu zadanej ilości sztuk
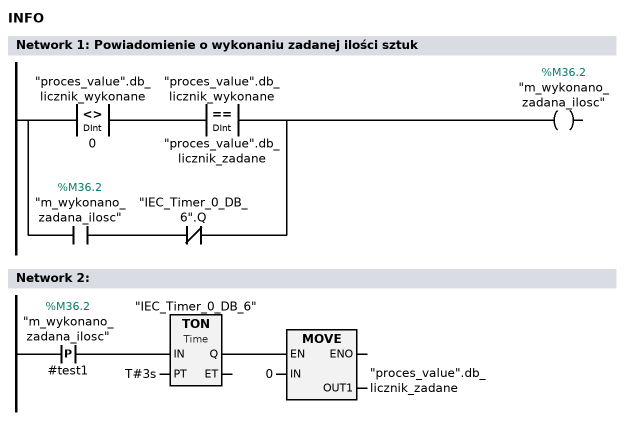
   RUNG wire#powerrail
      { S7_Templates := "SrcType := DInt" } NE_Contact(in1 := "proces_value".db_licznik_wykonane, in2 := 0)
      { S7_Templates := "SrcType := DInt" } EQ_Contact(in1 := "proces_value".db_licznik_wykonane, in2 := "proces_value".db_licznik_zadane)
      wire#w1
      Coil( "m_wykonano_zadana_ilosc" )
   END_RUNG
   RUNG wire#powerrail
      Contact( "m_wykonano_zadana_ilosc" )
      I_Contact( "IEC_Timer_0_DB_6".Q )
   END_RUNG wire#w1
   // the same network as SCL:
   "m_wykonano_zadana_ilosc" := (("proces_value".db_licznik_wykonane <> 0) AND ("proces_value".db_licznik_wykonane = "proces_value".db_licznik_zadane)) OR ("m_wykonano_zadana_ilosc" AND NOT "IEC_Timer_0_DB_6".Q);
END_REGION

REGION Network 2
   RUNG wire#powerrail
      P_Contact(operand := "m_wykonano_zadana_ilosc", bit := #test1)
      { S7_Templates := "time_type := Time" } "IEC_Timer_0_DB_6".TON(pt := T#3s, et =>)
      Move(in := 0, out1 => "proces_value".db_licznik_zadane)
   END_RUNG
   // the same network as SCL:
   #_w1 := "m_wykonano_zadana_ilosc" AND NOT #test1;   // rising edge of "m_wykonano_zadana_ilosc"
   #test1 := "m_wykonano_zadana_ilosc";
   "IEC_Timer_0_DB_6".TON(IN := #_w1, PT := T#3s);
   IF "IEC_Timer_0_DB_6".Q THEN "proces_value".db_licznik_zadane := 0; END_IF;
END_REGION

REGION Network 3: Info o Pauzie
END_REGION
END_FUNCTION

DATA_BLOCK "IEC_Timer_0_DB"   // DB1
{ S7_Optimized_Access := 'TRUE' }
// stored: AutoNumber true, DBAccessibleFromOPCUA true, InstanceOfName IEC_TIMER, OfSystemLibElement IEC_TIMER, OfSystemLibVersion 1.0
"IEC_TIMER"
   // VAR
   //    PT : Time;
   //    ET { ExternalWritable := 'False'} : Time;
   //    IN : Bool;
   //    Q { ExternalWritable := 'False'} : Bool;
   // END_VAR
BEGIN
END_DATA_BLOCK

DATA_BLOCK "IEC_Timer_0_DB_1"   // DB2
{ S7_Optimized_Access := 'TRUE' }
// stored: AutoNumber true, DBAccessibleFromOPCUA true, InstanceOfName IEC_TIMER, OfSystemLibElement IEC_TIMER, OfSystemLibVersion 1.0
"IEC_TIMER"
   // VAR
   //    PT : Time;
   //    ET { ExternalWritable := 'False'} : Time;
   //    IN : Bool;
   //    Q { ExternalWritable := 'False'} : Bool;
   // END_VAR
BEGIN
END_DATA_BLOCK

DATA_BLOCK "IEC_Timer_0_DB_10"   // DB18
{ S7_Optimized_Access := 'TRUE' }
// stored: AutoNumber true, DBAccessibleFromOPCUA true, InstanceOfName IEC_TIMER, OfSystemLibElement IEC_TIMER, OfSystemLibVersion 1.0
"IEC_TIMER"
   // VAR
   //    PT : Time;
   //    ET { ExternalWritable := 'False'} : Time;
   //    IN : Bool;
   //    Q { ExternalWritable := 'False'} : Bool;
   // END_VAR
BEGIN
END_DATA_BLOCK

DATA_BLOCK "IEC_Timer_0_DB_11"   // DB20
{ S7_Optimized_Access := 'TRUE' }
// stored: AutoNumber true, DBAccessibleFromOPCUA true, InstanceOfName IEC_TIMER, OfSystemLibElement IEC_TIMER, OfSystemLibVersion 1.0
"IEC_TIMER"
   // VAR
   //    PT : Time;
   //    ET { ExternalWritable := 'False'} : Time;
   //    IN : Bool;
   //    Q { ExternalWritable := 'False'} : Bool;
   // END_VAR
BEGIN
END_DATA_BLOCK

DATA_BLOCK "IEC_Timer_0_DB_12"   // DB21
{ S7_Optimized_Access := 'TRUE' }
// stored: AutoNumber true, DBAccessibleFromOPCUA true, InstanceOfName IEC_TIMER, OfSystemLibElement IEC_TIMER, OfSystemLibVersion 1.0
"IEC_TIMER"
   // VAR
   //    PT : Time;
   //    ET { ExternalWritable := 'False'} : Time;
   //    IN : Bool;
   //    Q { ExternalWritable := 'False'} : Bool;
   // END_VAR
BEGIN
END_DATA_BLOCK

DATA_BLOCK "IEC_Timer_0_DB_13"   // DB22
{ S7_Optimized_Access := 'TRUE' }
// stored: AutoNumber true, DBAccessibleFromOPCUA true, InstanceOfName IEC_TIMER, OfSystemLibElement IEC_TIMER, OfSystemLibVersion 1.0
"IEC_TIMER"
   // VAR
   //    PT : Time;
   //    ET { ExternalWritable := 'False'} : Time;
   //    IN : Bool;
   //    Q { ExternalWritable := 'False'} : Bool;
   // END_VAR
BEGIN
END_DATA_BLOCK

DATA_BLOCK "IEC_Timer_0_DB_14"   // DB23
{ S7_Optimized_Access := 'TRUE' }
// stored: AutoNumber true, DBAccessibleFromOPCUA true, InstanceOfName IEC_TIMER, OfSystemLibElement IEC_TIMER, OfSystemLibVersion 1.0
"IEC_TIMER"
   // VAR
   //    PT : Time;
   //    ET { ExternalWritable := 'False'} : Time;
   //    IN : Bool;
   //    Q { ExternalWritable := 'False'} : Bool;
   // END_VAR
BEGIN
END_DATA_BLOCK

DATA_BLOCK "IEC_Timer_0_DB_15"   // DB24
{ S7_Optimized_Access := 'TRUE' }
// stored: AutoNumber true, DBAccessibleFromOPCUA true, InstanceOfName IEC_TIMER, OfSystemLibElement IEC_TIMER, OfSystemLibVersion 1.0
"IEC_TIMER"
   // VAR
   //    PT : Time;
   //    ET { ExternalWritable := 'False'} : Time;
   //    IN : Bool;
   //    Q { ExternalWritable := 'False'} : Bool;
   // END_VAR
BEGIN
END_DATA_BLOCK

DATA_BLOCK "IEC_Timer_0_DB_16"   // DB25
{ S7_Optimized_Access := 'TRUE' }
// stored: AutoNumber true, DBAccessibleFromOPCUA true, InstanceOfName IEC_TIMER, OfSystemLibElement IEC_TIMER, OfSystemLibVersion 1.0
"IEC_TIMER"
   // VAR
   //    PT : Time;
   //    ET { ExternalWritable := 'False'} : Time;
   //    IN : Bool;
   //    Q { ExternalWritable := 'False'} : Bool;
   // END_VAR
BEGIN
END_DATA_BLOCK

DATA_BLOCK "IEC_Timer_0_DB_18"   // DB27
{ S7_Optimized_Access := 'TRUE' }
// stored: AutoNumber true, DBAccessibleFromOPCUA true, InstanceOfName IEC_TIMER, OfSystemLibElement IEC_TIMER, OfSystemLibVersion 1.0
"IEC_TIMER"
   // VAR
   //    PT : Time;
   //    ET { ExternalWritable := 'False'} : Time;
   //    IN : Bool;
   //    Q { ExternalWritable := 'False'} : Bool;
   // END_VAR
BEGIN
END_DATA_BLOCK

DATA_BLOCK "IEC_Timer_0_DB_2"   // DB3
{ S7_Optimized_Access := 'TRUE' }
// stored: AutoNumber true, DBAccessibleFromOPCUA true, InstanceOfName IEC_TIMER, OfSystemLibElement IEC_TIMER, OfSystemLibVersion 1.0
"IEC_TIMER"
   // VAR
   //    PT : Time;
   //    ET { ExternalWritable := 'False'} : Time;
   //    IN : Bool;
   //    Q { ExternalWritable := 'False'} : Bool;
   // END_VAR
BEGIN
END_DATA_BLOCK

DATA_BLOCK "IEC_Timer_0_DB_3"   // DB4
{ S7_Optimized_Access := 'TRUE' }
// stored: AutoNumber true, DBAccessibleFromOPCUA true, InstanceOfName IEC_TIMER, OfSystemLibElement IEC_TIMER, OfSystemLibVersion 1.0
"IEC_TIMER"
   // VAR
   //    PT : Time;
   //    ET { ExternalWritable := 'False'} : Time;
   //    IN : Bool;
   //    Q { ExternalWritable := 'False'} : Bool;
   // END_VAR
BEGIN
END_DATA_BLOCK

DATA_BLOCK "IEC_Timer_0_DB_4"   // DB5
{ S7_Optimized_Access := 'TRUE' }
// stored: AutoNumber true, DBAccessibleFromOPCUA true, InstanceOfName IEC_TIMER, OfSystemLibElement IEC_TIMER, OfSystemLibVersion 1.0
"IEC_TIMER"
   // VAR
   //    PT : Time;
   //    ET { ExternalWritable := 'False'} : Time;
   //    IN : Bool;
   //    Q { ExternalWritable := 'False'} : Bool;
   // END_VAR
BEGIN
END_DATA_BLOCK

DATA_BLOCK "IEC_Timer_0_DB_5"   // DB6
{ S7_Optimized_Access := 'TRUE' }
// stored: AutoNumber true, DBAccessibleFromOPCUA true, InstanceOfName IEC_TIMER, OfSystemLibElement IEC_TIMER, OfSystemLibVersion 1.0
"IEC_TIMER"
   // VAR
   //    PT : Time;
   //    ET { ExternalWritable := 'False'} : Time;
   //    IN : Bool;
   //    Q { ExternalWritable := 'False'} : Bool;
   // END_VAR
BEGIN
END_DATA_BLOCK

DATA_BLOCK "IEC_Timer_0_DB_6"   // DB7
{ S7_Optimized_Access := 'TRUE' }
// stored: AutoNumber true, DBAccessibleFromOPCUA true, InstanceOfName IEC_TIMER, OfSystemLibElement IEC_TIMER, OfSystemLibVersion 1.0
"IEC_TIMER"
   // VAR
   //    PT : Time;
   //    ET { ExternalWritable := 'False'} : Time;
   //    IN : Bool;
   //    Q { ExternalWritable := 'False'} : Bool;
   // END_VAR
BEGIN
END_DATA_BLOCK

DATA_BLOCK "IEC_Timer_0_DB_7"   // DB14
{ S7_Optimized_Access := 'TRUE' }
// stored: AutoNumber true, DBAccessibleFromOPCUA true, InstanceOfName IEC_TIMER, OfSystemLibElement IEC_TIMER, OfSystemLibVersion 1.0
"IEC_TIMER"
   // VAR
   //    PT : Time;
   //    ET { ExternalWritable := 'False'} : Time;
   //    IN : Bool;
   //    Q { ExternalWritable := 'False'} : Bool;
   // END_VAR
BEGIN
END_DATA_BLOCK

DATA_BLOCK "IEC_Timer_0_DB_8"   // DB13
{ S7_Optimized_Access := 'TRUE' }
// stored: AutoNumber true, DBAccessibleFromOPCUA true, InstanceOfName IEC_TIMER, OfSystemLibElement IEC_TIMER, OfSystemLibVersion 1.0
"IEC_TIMER"
   // VAR
   //    PT : Time;
   //    ET { ExternalWritable := 'False'} : Time;
   //    IN : Bool;
   //    Q { ExternalWritable := 'False'} : Bool;
   // END_VAR
BEGIN
END_DATA_BLOCK

DATA_BLOCK "IEC_Timer_0_DB_9"   // DB17
{ S7_Optimized_Access := 'TRUE' }
// stored: AutoNumber true, DBAccessibleFromOPCUA true, InstanceOfName IEC_TIMER, OfSystemLibElement IEC_TIMER, OfSystemLibVersion 1.0
"IEC_TIMER"
   // VAR
   //    PT : Time;
   //    ET { ExternalWritable := 'False'} : Time;
   //    IN : Bool;
   //    Q { ExternalWritable := 'False'} : Bool;
   // END_VAR
BEGIN
END_DATA_BLOCK

DATA_BLOCK "MC_Home_DB"   // DB11
// stored: AutoNumber true, DBAccessibleFromOPCUA true, InstanceOfName MC_Home, OfSystemLibElement MC_Home, OfSystemLibVersion 8.0
"MC_Home"
   // VAR_INPUT
   //    Axis : TO_Axis;
   //    Execute : Bool;
   //    Position : Real;
   //    Mode : Int;
   // END_VAR
   // VAR_OUTPUT
   //    Done : Bool;
   //    Busy : Bool;
   //    CommandAborted : Bool;
   //    Error : Bool;
   //    ErrorID : Word;
   //    ErrorInfo : Word;
   //    ReferenceMarkPosition : Real;
   // END_VAR
   // VAR
   //    FB_ID : DInt;
   // END_VAR
BEGIN
END_DATA_BLOCK

DATA_BLOCK "MC_MoveJog_DB"   // DB15
// stored: AutoNumber true, DBAccessibleFromOPCUA true, InstanceOfName MC_MoveJog, OfSystemLibElement MC_MoveJog, OfSystemLibVersion 8.0
"MC_MoveJog"
   // VAR_INPUT
   //    Axis : TO_SpeedAxis;
   //    JogForward : Bool;
   //    JogBackward : Bool;
   //    Velocity : Real;
   //    PositionControlled : Bool;
   // END_VAR
   // VAR_OUTPUT
   //    InVelocity : Bool;
   //    Busy : Bool;
   //    CommandAborted : Bool;
   //    Error : Bool;
   //    ErrorID : Word;
   //    ErrorInfo : Word;
   // END_VAR
   // VAR
   //    FB_ID : DInt;
   // END_VAR
BEGIN
END_DATA_BLOCK

DATA_BLOCK "MC_MoveJog_DB_1"   // DB16
// stored: AutoNumber true, DBAccessibleFromOPCUA true, InstanceOfName MC_MoveJog, OfSystemLibElement MC_MoveJog, OfSystemLibVersion 8.0
"MC_MoveJog"
   // VAR_INPUT
   //    Axis : TO_SpeedAxis;
   //    JogForward : Bool;
   //    JogBackward : Bool;
   //    Velocity : Real;
   //    PositionControlled : Bool;
   // END_VAR
   // VAR_OUTPUT
   //    InVelocity : Bool;
   //    Busy : Bool;
   //    CommandAborted : Bool;
   //    Error : Bool;
   //    ErrorID : Word;
   //    ErrorInfo : Word;
   // END_VAR
   // VAR
   //    FB_ID : DInt;
   // END_VAR
BEGIN
END_DATA_BLOCK

DATA_BLOCK "MC_MoveJog_DB_2"   // DB19
// stored: AutoNumber true, DBAccessibleFromOPCUA true, InstanceOfName MC_MoveJog, OfSystemLibElement MC_MoveJog, OfSystemLibVersion 8.0
"MC_MoveJog"
   // VAR_INPUT
   //    Axis : TO_SpeedAxis;
   //    JogForward : Bool;
   //    JogBackward : Bool;
   //    Velocity : Real;
   //    PositionControlled : Bool;
   // END_VAR
   // VAR_OUTPUT
   //    InVelocity : Bool;
   //    Busy : Bool;
   //    CommandAborted : Bool;
   //    Error : Bool;
   //    ErrorID : Word;
   //    ErrorInfo : Word;
   // END_VAR
   // VAR
   //    FB_ID : DInt;
   // END_VAR
BEGIN
END_DATA_BLOCK

DATA_BLOCK "MC_Power_DB"   // DB9
// stored: AutoNumber true, DBAccessibleFromOPCUA true, InstanceOfName MC_Power, OfSystemLibElement MC_Power, OfSystemLibVersion 8.0
"MC_Power"
   // VAR_INPUT
   //    Axis : TO_Axis;
   //    Enable : Bool;
   //    StartMode : Int;
   //    StopMode : Int;
   // END_VAR
   // VAR_OUTPUT
   //    Status : Bool;
   //    Busy : Bool;
   //    Error : Bool;
   //    ErrorID : Word;
   //    ErrorInfo : Word;
   // END_VAR
   // VAR
   //    FB_ID : DInt;
   // END_VAR
BEGIN
END_DATA_BLOCK

DATA_BLOCK "MC_Reset_DB"   // DB10
// stored: AutoNumber true, DBAccessibleFromOPCUA true, InstanceOfName MC_Reset, OfSystemLibElement MC_Reset, OfSystemLibVersion 8.0
"MC_Reset"
   // VAR_INPUT
   //    Axis : TO_Axis;
   //    Execute : Bool;
   //    Restart : Bool;
   // END_VAR
   // VAR_OUTPUT
   //    Done : Bool;
   //    Busy : Bool;
   //    Error : Bool;
   //    ErrorID : Word;
   //    ErrorInfo : Word;
   // END_VAR
   // VAR
   //    FB_ID : DInt;
   // END_VAR
BEGIN
END_DATA_BLOCK
